// SIMATIC STEP 7 (V5.x) project Odbieranie_Kolbusy_Rob
// CPU: CPU 313C
// CPU: CPU 315-2 PN/DP
// CPU: CPU 315-2 DP
// CPU: CPU 315-2 DP
// CPU: CPU 315-2 DP
// station: Hardware
// station: Bandy
// station: P_ADR_BUS
// station: P_ADR_BUS
// station: Hardware
// station: Foliarka
// station: Hardware
// station: Odbieranie
// station: P_ADR_BUS
// station: Hardware
// station: Shuttle
// station: P_ADR_BUS
// station: P_ADR_BUS
// station: Hardware
// station: W_Help_PLC_TEST
// station: _S7H_BUSSYSTEM_CT
// station: P_ADR_BUS
// station: Configuration
// program: S7 Program
// program: S7 Program
// program: S7 Program
// program: S7 Program
// program: S7 Program(15)
// program: S7_Program_Band_Stary
// program: S7 _Bandy_1_Krew

SYMBOL_TABLE
"RUNNING_PROG"	DB 12	DB 12	// RUNNING PROGRAMME
"EDITING_PROG"	DB 13	DB 13	// EDITING PROGRAMME
"PROG_1_DATA"	DB 21	DB 21	// PROGRAMME 1
"PROG_2_DATA"	DB 22	DB 22	// PROGRAMME 2
"PROG_3_DATA"	DB 23	DB 23	// PROGRAMME 3
"PROG_4_DATA"	DB 24	DB 24	// PROGRAMME 4
"PROG_5_DATA"	DB 25	DB 25	// PROGRAMME 5
"PROG_6_DATA"	DB 26	DB 26	// PROGRAMME 6
"PROG_7_DATA"	DB 27	DB 27	// PROGRAMME 7
"PROG_8_DATA"	DB 28	DB 28	// PROGRAMME 8
"PROG_9_DATA"	DB 29	DB 29	// PROGRAMME 9
"INTERFACE_AREA"	DB 30	DB 30	// INTERFACE AREA
"MPI_GD"	DB 100	DB 100	// Blok wymiany danych po mpi
"CONTROL"	FC 1	FC 1	// CONTROL
"SAFETY_STOP"	FC 3	FC 3	// SAFETY STOP
"LAMP_TEST"	FC 4	FC 4	// LAMP TEST
"SIGNAL_OUT_CONVEYORS"	FC 5	FC 5	// EXTERNAL SIGNAL OUTPUT
"AUTOMATIC"	FC 10	FC 10	// AUTO / SEMIAUTO CHOICE
"PROGRAMME_CHOICE"	FC 11	FC 11	// START WRAPPING SEQUENCE AND PROGRAMME CHOICE
"MOTOR_TO_CLUTCH"	FC 12	FC 12	// MOTOR TO CLUTCH, SEQUENCE
"RESET_SEQ"	FC 13	FC 13	// RESET SEQUENCE
"CONVEYORING_SEQUENCE"	FC 14	FC 14	// CONVEYORING SEQUENCE
"WRAPPING_SEQUENCE"	FC 15	FC 15	// AUTOMATIC SEQUENCE
"START_AFTER_90_INFEED"	FC 16	FC 16	// START SEQ IN WRAPPING SEQ, 90 DEGREE INFEED
"90_DEGREE_INFEED"	FC 17	FC 17	// 90 DEGREE INFEED
"90_DEGREE_OUTFEED"	FC 18	FC 18	// 90 DEGREE OUTFEED
"TURN_TO/FROM_90_DEG"	FC 19	FC 19	// TURN TABLE TO/FROM 90 DEGREE
"PALLET_POS"	FC 21	FC 21	// PALLET POSITION, LENGTH MEASURE, OPTION
"TURNTABLE"	FC 22	FC 22	// TURNTABLE
"CARRIAGE"	FC 23	FC 23	// CARRIAGE
"TOPPLATE"	FC 24	FC 24	// TOPPLATE, OPTION
"FILM_FEED_SYSTEM"	FC 25	FC 25	// FILM FEED SYSTEM
"FILM_HOLDING_DEVICE"	FC 26	FC 26	// VALVES
"CUTTING_UNIT"	FC 27	FC 27	// VALVES
"HOT_AIR_WELDING"	FC 28	FC 28	// HOT AIR WELDING, OPTION
"WELDING"	FC 29	FC 29	// WELDING
"TURNTABLE_COUNTERS"	FC 32	FC 32	// TURNTABLE COUNTERS TO POSITION
"CARRIAGE_COUNTERS"	FC 33	FC 33	// CARRIAGE COUNTERS TO POSITION
"COUNTERS"	FC 34	FC 34	// COUNTERS
"CONVEYOR_1"	FC 71	FC 71	// CONVEYOR POS.1
"CONVEYOR_2"	FC 72	FC 72	// CONVEYOR AND TURN TABLE POS.2
"CONVEYOR_3"	FC 73	FC 73	// CONVEYOR POS.3
"CONVEYOR_4"	FC 74	FC 74	// CONVEYOR POS.4
"CONVEYOR_6"	FC 76	FC 76	// CONVEYOR POS.6
"CONVEYOR_7"	FC 77	FC 77	// CONVEYOR POS.7
"CONV_2"	FC 92	FC 92	// Stary przenosnik 2
"Komunikacja_GD"	FC 100	FC 100	// Komunikacja szafa foliarka
"DISPLAY_HANDLING"	FC 110	FC 110	// DISPLAY HANDLING
"MANUAL_MODE"	FC 111	FC 111	// TO RUN MACHINE IN MANUAL MODE
"ALARM"	FC 120	FC 120	// ALARM
"E 0.0"	I 0.0	BOOL	// CONTROLL VOLTAGE ON
"E 0.1"	I 0.1	BOOL	// MAIN VOLTAGE ON
"E 0.2"	I 0.2	BOOL	// TRANSDUCER TURNTABLE MOTOR FORWARD POSITION
"E 0.3"	I 0.3	BOOL	// TRANSDUCER TURNTABLE MOTOR REVERSE POSITION
"E 0.4"	I 0.4	BOOL	// TRANSDUCER TURNTABLE IN STARTPOSITION
"E 0.5"	I 0.5	BOOL	// TRANSDUCER TURNTABLE ROTATION
"E 0.6"	I 0.6	BOOL	// TRANSDUCER CARRIAGE ROTATION
"E 0.7"	I 0.7	BOOL	// TRANSDUCER TURNTABLE IN 90 DEGREE POSITION(OPTION)
"E 1.0"	I 1.0	BOOL	// TRANSDUCER PUSHER 90 DEGREE IN OUTER POSITION(OPTION)
"E 1.1"	I 1.1	BOOL	// PHOTOCELL INFEEDING START CONVEYOR
"E 1.2"	I 1.2	BOOL	// PHOTOCELL STOP INFEEDING
"E 1.3"	I 1.3	BOOL	// PHOTOCELL OUTFEEDING CONVEYOR NOT FULL(OPTION)
"E 1.5"	I 1.5	BOOL	// PHOTOCELL INDICATION PALLET 1/2 OR 1/1 SIZE OR SAFTEY
"E 1.6"	I 1.6	BOOL	// PHOTOCELL SAFETY PALLET SIZE / LENGTH MEASURE, INFEED SIDE
"E 1.7"	I 1.7	BOOL	// PHOTOCELL SAFETY PALLET SIZE / LENGTH MEASURE, OUTFEED SIDE
"E 4.0"	I 4.0	BOOL	// PB CONVEYOR 1 FORWARD(OPTION)
"E 4.1"	I 4.1	BOOL	// PB CONVEYOR 1 BACKWARD(OPTION)
"E 4.2"	I 4.2	BOOL	// PB CONVEYOR 2 FORWARD(OPTION)
"E 4.3"	I 4.3	BOOL	// PB CONVEYOR 2 BACKWARD(OPTION)
"E 4.4"	I 4.4	BOOL	// PB TURNNTABLE 2 TURN FORWARD(OPTION)
"E 4.5"	I 4.5	BOOL	// PB TURNNTABLE 2 TURN BACKWARD(OPTION)
"E 4.6"	I 4.6	BOOL	// PB CONVEYOR 3 FORWARD(OPTION)
"E 4.7"	I 4.7	BOOL	// PB CONVEYOR 3 BACKWARD(OPTION)
"E 5.0"	I 5.0	BOOL	// PB CONVEYOR 4 FORWARD
"E 5.1"	I 5.1	BOOL	// PB CONVEYOR 4 BACKWARD
"E 5.4"	I 5.4	BOOL	// PB CONVEYOR 6 FORWARD
"E 5.5"	I 5.5	BOOL	// PB CONVEYOR 6 BACKWARD
"E 5.6"	I 5.6	BOOL	// PB CONVEYOR 7 FORWARD
"E 5.7"	I 5.7	BOOL	// PB CONVEYOR 7 BACKWARD
"E 8.0"	I 8.0	BOOL	// Q PROTECTION TOP PLATE
"E 8.1"	I 8.1	BOOL	// TOPPLATE UPPER LIMIT
"E 8.2"	I 8.2	BOOL	// TOPPLATE LOWER LIMIT
"E 8.3"	I 8.3	BOOL	// TRANSDUCER TOP PLATE AGAINST GOODS
"E 8.5"	I 8.5	BOOL	// PUSH BUTTON, TOPPLATE UPWARDS
"E 8.6"	I 8.6	BOOL	// PUSH BUTTON, TOPPLATE DOWNWARDS
"E 9.0"	I 9.0	BOOL	// LS PALLET ON CONVEYOR 3(OPTION)
"E 9.1"	I 9.1	BOOL	// LS GAP MONITORING TURNTABLE CONVEYOR 3(OPTION)
"E 9.2"	I 9.2	BOOL	// LS PALLET ON CONVEYOR 1(OPTION)
"E 9.3"	I 9.3	BOOL	// LS PALLET ON CONVEYOR 2(OPTION)
"E 9.4"	I 9.4	BOOL	// AS TURN TABLE IN 0 DEGREES(OPTION)
"E 9.5"	I 9.5	BOOL	// MS SAFETY TURN TABLE IN 0 DEGREES(OPTION)
"E 9.6"	I 9.6	BOOL	// AS TURN TABLE IN 90 DEGREES(OPTION)
"E 9.7"	I 9.7	BOOL	// MS SAFETY TURN TABLE IN 90 DEGREES(OPTION)
"E 12.0"	I 12.0	BOOL	// MSI_FAULT SIGNAL
"E 12.1"	I 12.1	BOOL	// S1-S4 LIGHT  GRATING
"E 12.2"	I 12.2	BOOL	// 1.1-2.2 MSI DOORS
"E 12.3"	I 12.3	BOOL	// MSI MUTING IS ON
"E 12.4"	I 12.4	BOOL	// SIGNAL MUTING FAILURE
"E 12.5"	I 12.5	BOOL	// ALARM MUTING LAMP DEFECT
"E 12.6"	I 12.6	BOOL	// MSI RESTART BLOCKED
"E 12.7"	I 12.7	BOOL	// MSI STATE OF SAFETY OUTPUT
"E 13.0"	I 13.0	BOOL	// LS MUTING PHOTOCELL ON INFEEDING SIDE
"E 13.1"	I 13.1	BOOL	// LS MUTING PHOTOCELL ON OUTFEEDING SIDE
"E 13.2"	I 13.2	BOOL	// PB ACTIVATE SAFETY CIRCUIT
"E 13.3"	I 13.3	BOOL	// LS PALLET ON CONVEYOR 4
"E 13.4"	I 13.4	BOOL	// LS GAP MONITORING TURNTABLE CONVEYOR 6
"E 13.5"	I 13.5	BOOL	// LS PALLET ON CONVEYOR 6
"E 13.6"	I 13.6	BOOL	// LS PALLET ON CONVEYOR 7
"E 16.0"	I 16.0	BOOL	// FREQ.CONVERTER CONVEYOR 1 FAULT
"E 16.1"	I 16.1	BOOL	// FREQ.CONVERTER CONVEYOR 2 FAULT
"E 16.2"	I 16.2	BOOL	// FREQ.CONVERTER CONVEYOR 3 FAULT
"E 16.3"	I 16.3	BOOL	// FREQ.CONVERTER CONVEYOR 4 FAULT
"E 16.4"	I 16.4	BOOL	// Q MOTOR PROTECTION TURN TABLE 2 FAULT
"E 16.5"	I 16.5	BOOL	// Q MOTOR PROTECTION CONVEYOR 6 FAULT
"E 16.6"	I 16.6	BOOL	// Q MOTOR PROTECTION CONVEYOR 7 FAULT
"E 17.0"	I 17.0	BOOL	// MAIN CONTACTOR 1 ON
"E 17.1"	I 17.1	BOOL	// MAIN CONTACTOR 2 ON
"E 124.0"	I 124.0	BOOL	// PB AUTOMATIC ON
"E 124.1"	I 124.1	BOOL	// PB SEMIAUTOMATIC ON
"E 124.2"	I 124.2	BOOL	// PB STOP
"E 124.3"	I 124.3	BOOL	// PB MACHINE TO HOME POSITION / RESET
"E 124.4"	I 124.4	BOOL	// PB START SELECT WRAPPING PROGRAM
"E 124.5"	I 124.5	BOOL	// PB TURNTABLE CONVEYOR FORWARD, A
"E 124.6"	I 124.6	BOOL	// PB TURNTABLE CONVEYOR REVERSE, B
"E 124.7"	I 124.7	BOOL	// FILM CONSUMPTION (OPTION)
"E 125.0"	I 125.0	BOOL	// AS TRANSDUCER FILM END
"E 125.1"	I 125.1	BOOL	// MS CARRIAGE UPPER LIMIT
"E 125.2"	I 125.2	BOOL	// MS CARRIAGE LOWER LIMIT
"E 125.3"	I 125.3	BOOL	// AS CARRIAGE STARTPOSITION
"E 125.4"	I 125.4	BOOL	// LS PHOTOCELL PALLETHEIGHT
"E 125.5"	I 125.5	BOOL	// MS CARRIAGE CRUTSH PROTECTION
"E 125.6"	I 125.6	BOOL	// AS CUTTING DEVICE REVERSE POSITION
"E 125.7"	I 125.7	BOOL	// AS CUTTING DEVICE 1/2 - REVERSE POSITION
"E 126.0"	I 126.0	BOOL	// PROGRAMME SELECTION REMOTE COMTROLLED, BIN 1
"E 126.1"	I 126.1	BOOL	// PROGRAMME SELECTION REMOTE COMTROLLED, BIN 2
"E 126.2"	I 126.2	BOOL	// PROGRAMME SELECTION REMOTE COMTROLLED, BIN 4
"E 126.3"	I 126.3	BOOL	// FREQ.CONVERTER film motor
"E 126.4"	I 126.4	BOOL	// EXT> CONEYOR RUN IN IS RUNNING
"E 126.5"	I 126.5	BOOL	// EXT> PALLET IS READY FOR RUN IN TO CONVEYOR 1
"E 126.6"	I 126.6	BOOL	// FREQ.CONVERTER CARRIAGE FAULT
"E 126.7"	I 126.7	BOOL	// FERG.COVERTER TURN TABLE-CONVEYOR FAULT
"M 70.0"	M 70.0	BOOL	// FC71 -CONVEYOR POS.1 LOCKING
"M 70.1"	M 70.1	BOOL	// FC71 -CONVEYOR POS.1 FU FAULT
"M 70.2"	M 70.2	BOOL	// FC71 -CONVEYOR POS.1 RUN IN
"M 70.3"	M 70.3	BOOL	// FC71 -CONVEYOR POS.1 OCCUPIED
"M 70.4"	M 70.4	BOOL	// FC71 -CONVEYOR POS.1 RUN OUT
"M 70.5"	M 70.5	BOOL	// FC71 -CONVEYOR POS.1 FORWARD
"M 70.6"	M 70.6	BOOL	// FC71 -CONVEYOR POS.1 BACKWARD
"M 70.7"	M 70.7	BOOL	// FC71 -CONVEYOR POS.1 RUNTIME
"M 72.0"	M 72.0	BOOL	// FC72 -CONVEYOR POS.2 LOCKING
"M 72.1"	M 72.1	BOOL	// FC72 -CONVEYOR POS.2 FU FAULT
"M 72.2"	M 72.2	BOOL	// FC72 -CONVEYOR POS.2 RUN IN
"M 72.3"	M 72.3	BOOL	// FC72 -CONVEYOR POS.2 OCCUPIED
"M 72.4"	M 72.4	BOOL	// FC72 -CONVEYOR POS.2 RUN OUT
"M 72.5"	M 72.5	BOOL	// FC72 -CONVEYOR POS.2 FORWARD
"M 72.6"	M 72.6	BOOL	// FC72 -CONVEYOR POS.2 BACKWARD
"M 72.7"	M 72.7	BOOL	// FC72 -CONVEYOR POS.2 RUNTIME
"M 74.0"	M 74.0	BOOL	// FC72 -TURN TABLE POS.2 LOCKING
"M 74.1"	M 74.1	BOOL	// FC72 -TURN TABLE POS.2 MOTOR FAULT
"M 74.2"	M 74.2	BOOL	// FC72 -TURN TABLE POS.2 RUN TO 0DEG
"M 74.3"	M 74.3	BOOL	// FC72 -TURN TABLE POS.2 SPARE
"M 74.4"	M 74.4	BOOL	// FC72 -TURN TABLE POS.2 RUN TO 90DEG
"M 74.5"	M 74.5	BOOL	// FC72 -TURN TABLE POS.2 TURN FORWARD
"M 74.6"	M 74.6	BOOL	// FC72 -TURN TABLE POS.2 TURN BACKWARD
"M 74.7"	M 74.7	BOOL	// FC72 -TURN TABLE POS.2 RUNTIME
"M 75.0"	M 75.0	BOOL	// FC72 -TURN TABLE POS.2 GAP FAULT
"M 75.1"	M 75.1	BOOL	// FC72 -TURN TABLE POS.2 SAFETY SWITCH FAULT
"M 76.0"	M 76.0	BOOL	// FC73 -CONVEYOR POS.3 LOCKING
"M 76.1"	M 76.1	BOOL	// FC73 -CONVEYOR POS.3 FU FAULT
"M 76.2"	M 76.2	BOOL	// FC73 -CONVEYOR POS.3 RUN IN
"M 76.3"	M 76.3	BOOL	// FC73 -CONVEYOR POS.3 OCCUPIED
"M 76.4"	M 76.4	BOOL	// FC73 -CONVEYOR POS.3 RUN OUT
"M 76.5"	M 76.5	BOOL	// FC73 -CONVEYOR POS.3 FORWARD
"M 76.6"	M 76.6	BOOL	// FC73 -CONVEYOR POS.3 BACKWARD
"M 76.7"	M 76.7	BOOL	// FC73 -CONVEYOR POS.3 RUNTIME
"M 78.0"	M 78.0	BOOL	// FC74 -CONVEYOR POS.4 LOCKING
"M 78.1"	M 78.1	BOOL	// FC74 -CONVEYOR POS.4 FU FAULT
"M 78.2"	M 78.2	BOOL	// FC74 -CONVEYOR POS.4 RUN IN
"M 78.3"	M 78.3	BOOL	// FC74 -CONVEYOR POS.4 OCCUPIED
"M 78.4"	M 78.4	BOOL	// FC74 -CONVEYOR POS.4 RUN OUT
"M 78.5"	M 78.5	BOOL	// FC74 -CONVEYOR POS.4 FORWARD
"M 78.6"	M 78.6	BOOL	// FC74 -CONVEYOR POS.4 BACKWARD
"M 78.7"	M 78.7	BOOL	// FC74 -CONVEYOR POS.4 RUNTIME
"M 79.0"	M 79.0	BOOL	// FC74 -ONE SHOT RUN IN POS.4
"M 80.0"	M 80.0	BOOL	// FC76 -CONVEYOR POS.6 LOCKING
"M 80.1"	M 80.1	BOOL	// FC76 -CONVEYOR POS.6 MOTOR FAULT
"M 80.2"	M 80.2	BOOL	// FC76 -CONVEYOR POS.6 RUN IN
"M 80.3"	M 80.3	BOOL	// FC76 -CONVEYOR POS.6 OCCUPIED
"M 80.4"	M 80.4	BOOL	// FC76 -CONVEYOR POS.6 RUN OUT
"M 80.5"	M 80.5	BOOL	// FC76 -CONVEYOR POS.6 FORWARD
"M 80.6"	M 80.6	BOOL	// FC76 -CONVEYOR POS.6 BACKWARD
"M 80.7"	M 80.7	BOOL	// FC76 -CONVEYOR POS.6 RUNTIME
"M 82.0"	M 82.0	BOOL	// FC77 -CONVEYOR POS.7 LOCKING
"M 82.1"	M 82.1	BOOL	// FC77 -CONVEYOR POS.7 MOTOR FAULT
"M 82.2"	M 82.2	BOOL	// FC77 -CONVEYOR POS.7 RUN IN
"M 82.3"	M 82.3	BOOL	// FC77 -CONVEYOR POS.7 OCCUPIED
"M 82.4"	M 82.4	BOOL	// FC77 -CONVEYOR POS.7 RUN OUT
"M 82.5"	M 82.5	BOOL	// FC77 -CONVEYOR POS.7 FORWARD
"M 82.6"	M 82.6	BOOL	// FC77 -CONVEYOR POS.7 BACKWARD
"M 82.7"	M 82.7	BOOL	// FC77 -CONVEYOR POS.7 RUNTIME
"RAMP_STOP_IN_HOME_POS"	M 92.3	BOOL	// HELPMEMORY FOR RAMP DOWN BEFORE STOP IN HOME POS.
"NO_SEQ_RUNNING"	M 96.0	BOOL	// NO SEQUENCE RUNNING
"WRAPP_NOT_RUNNING"	M 96.1	BOOL	// WRAPPING PROGRAMME NOT RUNNING
"WRAPP90_NOT_RUNNING"	M 96.2	BOOL	// WRAPPING PROGRAMME FROM 90 INFEEDING NOT RUNNING
"MOTOR_TO_CLUTCH_NOT_RUN"	M 96.3	BOOL	// SEQUENCE MOTOR TO CLUTCH NOT RUNNING
"OK_FROM_TP"	M 96.5	BOOL	// TOPPLATE NOT AGAINST PALLET
"RESET_NOT_RUNNING"	M 97.2	BOOL	// RESET NOT RUNNING, MACHINE TO INITIAL POSITION
"CONVEYORING_NOT_RUNNING"	M 97.3	BOOL	// SEQUENCE CONVEYORING NOT RUNNING
"SEQ_90_INFEED_NOT_RUN"	M 97.4	BOOL	// SEQUENCE 90 DEGREE INFEEDING NOT RUNNING
"SEQ_90_OUTFEED_NOT_RUN"	M 97.5	BOOL	// SEQUENCE 90 DEGREE OUTFEEDING NOT RUNNING
"SEQ_TO/FROM_90_DEGREE"	M 97.6	BOOL	// SEQUENCE TO/FROM 90 DEGREE NOT RUNNING
"JUMP_RESET"	M 97.7	BOOL	// CONDITION TO JUMP TO RESET PROGREMME
"PULSE_PROG_REGISTER"	M 98.0	BOOL	// PULSE TO PROGRAMME REGISTER
"NO_PROG_RUNNING"	M 98.1	BOOL	// NO PROGRAMME RUNNING
"JUMP_RESET_MW"	M 98.2	BOOL	// CONDITION TO JUMP TO RESET MW, PUT ZERO TO MEM
"PULSE_RESET"	M 98.3	BOOL	// PULSE RESET
"RESET_HOLD"	M 98.4	BOOL	// PREVENT RESTART RESET SEQUENCE
"PROG_5_CHOICED"	M 98.5	BOOL	// PROGRAM 5 FILM AND OUT BACK TO STRAPPER
"PROG_4_CHOICED"	M 98.7	BOOL	// PROGRAMME 4, CONVEYORING THROUGH
"HELP_TO_M98.0"	M 99.0	BOOL	// HELP TO "PULSE_PROGRAMME REGISTER"
"HELP_TO_M98.2"	M 99.2	BOOL	// HELP TO "JUMP_RESET_MW"
"HELP_TO_M98.3"	M 99.3	BOOL	// HELP TO "PULSE_RESET"
"AUTO"	M 102.0	BOOL	// AUTOMATC MODE
"PULSE_FILMCONS"	M 103.0	BOOL	// PULSE TO COUNT UP FILM CONSUMPTION
"HELP_PULSE_FILMCONS"	M 103.1	BOOL	// HELP PULSE FILM CONSUMPTION
"COUNT_WRAP"	M 103.2	BOOL	// COUNT NUMBERS OF WRAPPING
"HELP_COUNT_WRAP"	M 103.3	BOOL	// HELP TO COUNT NUMBERS OF WRAPPING
"HELP_COUNT_FILMCON"	M 103.4	BOOL	// HELP TO COUNT FILN CONSUMPTION
"ST.MOT1"	M 118.1	BOOL	// START SEQUENCE MOTOR TO CLUTCH
"ST.MOT2"	M 118.2	BOOL	// MOTOR FORWARDS
"ST.MOT3"	M 118.3	BOOL	// MOTOR FWD SPEED 1
"ST.MOT4"	M 118.4	BOOL	// MOTOR REV SPEED 1
"ST.MOT5"	M 118.5	BOOL	// MOTOR STOP
"ST.MOT6"	M 118.6	BOOL	// TURNTABLE MOTOR IN FORWARD POSITION
"RESET_STEP1"	M 120.1	BOOL	// MOTOR BACKWARDS
"RESET_STEP2"	M 120.2	BOOL	// MOTOR SPEED 2
"RESET_STEP3"	M 120.3	BOOL	// SYNC TURNTABLE
"RESET_STEP4"	M 120.4	BOOL	// MOTOR SPEED 1
"RESET_STEP5"	M 120.5	BOOL	// MOTOR STOP, TO CLUTCH
"RESET_STEP6"	M 120.6	BOOL	// MOTOR FORWARD POSITION
"RESET_STEP7"	M 120.7	BOOL	// CARRIAGE UP
"RESET_STEP8"	M 121.0	BOOL	// CARRIAGE DOWN
"RESET_STEP9"	M 121.1	BOOL	// CARRIAGE IN POSITION
"RESET_STEP10"	M 121.2	BOOL	// RESET CYCLE FINISHED
"TPC.RES"	M 124.0	BOOL	// RESETING CONVEYOR CYCLE
"ST.TP1"	M 124.1	BOOL	// CONVEYOR INFEEDING
"ST.TP2"	M 124.2	BOOL	// OK TO START INFEEDING
"ST.TP3"	M 124.3	BOOL	// INFEEDING STOP
"ST.TP4"	M 124.4	BOOL	// OUTFEEDING REQUEST
"ST.TP5"	M 124.5	BOOL	// CONVEYOR START OUTFEEDING
"ST.TP6"	M 124.6	BOOL	// CONVEYOR OUTFEEDING
"ST.TP00"	M 124.7	BOOL	// CONVEYOR CYCLE NOT RUNNING
"FROM_LEFT"	M 126.1	BOOL	// CONVEYORING IN FROM LEFT TO RIGHT, OR FROM LEFT OUT 90
"TO_LEFT"	M 126.2	BOOL	// CONVEYORING OUT FROM RIGHT TO LEFT, OR IN 90 OUT LEFT
"FROM_RIGHT"	M 126.3	BOOL	// CONVEYORING IN FROM RIGHT TO LEFT, OR FROM RIGHT OUT 90
"TO_RIGHT"	M 126.4	BOOL	// CONVEYORING OUT FROM LEFT TO RIGHT, OR IN 90 OUT RIGHT
"FROM_90_D"	M 126.5	BOOL	// CONVEYORING IN FROM 90 DEGREE
"TO_90_D"	M 126.6	BOOL	// CONVEYORING OUT TO 90 DEGREE
"S15_SAFTY_HELP"	M 126.7	BOOL	// HELP MEM, PHOTOCELL SAFETY PALLET SIZE, TO LONG INFEEDING, 90 DEG
"PULSE_TIME_50"	M 132.0	BOOL	// BIT FOR TIME PULSE, T 50
"PALLET_INFEED"	M 132.1	BOOL	// BIT PALLET INFEEDING
"CNT_SIZE_RUN"	M 132.2	BOOL	// COUNTING SIZE IS RUNNING
"START_CNT_SIZE"	M 132.3	BOOL	// START PULSE COUNTING SIZE
"CNT_STOP_TIME"	M 132.4	BOOL	// COUNTING STOP TIME
"START_CNT_STOP_TIME"	M 132.5	BOOL	// PULSE START COUNT STOP TIME
"CNT_SIZE"	M 132.6	BOOL	// BIT FOR TIME COUNTING SIZE
"STOP_COUNTING"	M 132.7	BOOL	// BIT FOR STOP TIME COUNTING
"STOP_PALLET"	M 133.0	BOOL	// HELP BIT STOP PALLET
"STOP_SP"	M 133.6	BOOL	// STOP NEW STARTPULSE
"STOP_PST"	M 133.7	BOOL	// STOP NEW PULSE STOP TIME
"LOCK-U1"	M 134.0	BOOL	// LOCKING TURNTABLE
"TT_SPEED_LOW_FWD"	M 134.1	BOOL	// TURNTABLE SPEED LOW
"TT_SPEED_MIDDLE_FWD"	M 134.2	BOOL	// TURNTABLE SPEED MIDDLE
"TT_SPEED_HIGH"	M 134.3	BOOL	// TURNTABLE SPEED HIGH
"TT_SPEED_CONV"	M 134.4	BOOL	// CONVEYOR SPEED
"CONV_LEFT"	M 134.5	BOOL	// CONVEYOR LEFT
"CONV_RIGHT"	M 134.6	BOOL	// CONVEYOR RIGHT
"TT_FREQ_CONV_RUN"	M 134.7	BOOL
"TT_HELP_SPEED"	M 135.0	BOOL	// TURNTABLE SPEED MIDDLE OR HIGH
"TT_SPEED_LOW_REV"	M 135.1	BOOL	// TURNTABLE SPEED LOW
"TT_SPEED_MIDDLE_REV"	M 135.2	BOOL	// TURNTABLE SPEED MIDDLE
"TT_OK_TO_START"	M 135.3	BOOL	// TURNTABLE MOTOR STANDS STILL, OK TO START
"U1_INCREASE_COARSE"	M 135.4	BOOL	// TURNTABLE SPEED INCREASE COARSE
"U1_REDUSE_COARSE"	M 135.5	BOOL	// TURNTABLE SPEED REDUSE COARSE
"U1_INCREASE_FINE"	M 135.6	BOOL	// TURNTABLE SPEED INCREASE FINE
"U1_REDUSE_FINE"	M 135.7	BOOL	// TURNTABLE SPEED REDUSE FINE
"LOCK-U3"	M 136.0	BOOL	// LOCKING CARRIAGE
"CARR_SPEED_UP"	M 136.1	BOOL	// CARRIAGE SPEED UP
"CARR_SPEED_DOWN"	M 136.2	BOOL	// CARRIAGE SPEED DOWN
"CARR_HIGH_SPEED"	M 136.3	BOOL	// CARRIAGE SPEED HIGH
"CARR_RESET_SPEED"	M 136.4	BOOL	// CARRIAGE SPEED RESET
"CARR_UPWARDS"	M 136.5	BOOL	// CARRIAGE UP
"CARR_DOWNWARDS"	M 136.6	BOOL	// CARRIAGE DOWN
"CARR_FREQ_CONV_RUN"	M 136.7	BOOL
"CARR_OK_TO_START"	M 137.3	BOOL	// CARRIAGE MOTOR STANDS STILL, OK TO START
"U3_INCREASE_COARSE"	M 137.4	BOOL	// CARRIAGE SPEED INCREASE COARSE
"U3_REDUSE_COARSE"	M 137.5	BOOL	// CARRIAGE SPEED REDUSE COARSE
"U3_INCREASE_FINE"	M 137.6	BOOL	// CARRIAGE SPEED INCREASE FINE
"U3_REDUSE_FINE"	M 137.7	BOOL	// CARRIAGE SPEED REDUSE FINE
"WITH_TOPPLATE"	M 138.0	BOOL	// WRAPPING PROGRAMME WITH TOPPLATE
"TP_SAFETY_STOP_D"	M 138.1	BOOL	// TOPPLATE, SAFETY STOP DOWNWARDS
"HELP_TP_DOWNWARDS"	M 138.2	BOOL	// MEMORY TOPPLATE DOWNWARDS
"HELP_TP_UPWARDS"	M 138.3	BOOL	// MEMORY TOPPLATE UPWARDS
"LOCK-U2"	M 140.0	BOOL	// LOCKING FILM MOTOR
"FILM_FREE"	M 140.1	BOOL	// OK TO RUN FILMMOTOR
"PULSE_FFS"	M 140.2	BOOL	// PULES TO INCREASE FILMFEED VALUE
"CLUTCH_ON_CUT"	M 140.3	BOOL	// CLUTCH ON, CUTTING FILM
"ST.FF1"	M 141.1	BOOL	// INCREASE FILMFEED VALUE
"ST.FF2"	M 141.2	BOOL	// REDUCE FILMFEED VALUE
"ST.FF3"	M 141.3	BOOL	// REDUCE FILMFEED VALUE WITH FILMTENSION
"ST.FF4"	M 141.4	BOOL	// REDUCE FILMFEED AFTER CLUTCH OFF
"LOCK_VALVE"	M 142.0	BOOL	// LOCKING SOLENOIDS
"LOCK_H_A_WELD"	M 146.0	BOOL	// LOCKING HOT AIR WELDING
"HELP_TO_M146.2"	M 146.1	BOOL	// HELP TO "H A WELD START"
"H_A_WELD_START"	M 146.2	BOOL	// IMPULS HOT AIR WELDING START
"H_A_W_HEATING"	M 146.3	BOOL	// HOT AIR WELDING, HEATING
"H_A_WELD_ON"	M 146.5	BOOL	// HOT AIR WELDING ON
"H_A_WELD_FIN"	M 146.6	BOOL	// HOT AIR WELDING FINISHED
"TURNTABLE_COUNT_MEM"	M 160.0	BOOL	// COUNT UP TURNTABLE POSITION
"HELP_PF_TURNTABLE_C"	M 160.1	BOOL	// POSITIVE FLANK TURNTABLE COUNTER
"HELP_NF_TURNTABLE_C"	M 160.2	BOOL	// NEGATIVE FLANK TURNTABLE COUNTER
"OK_COMPARE"	M 160.3	BOOL
"MEM_BW"	M 160.4	BOOL	// HELP MEMORY THEN BOTTOMWRAPPING RUNNING
"MEM_TW"	M 160.5	BOOL	// HELP MEMORY THEN TOPWRAPPING RUNNING
"HELP_PF_TURNT_IN_POS"	M 160.6	BOOL	// POSITIVE FLANK TURNTABLE COUNTER
"BW_READY"	M 162.1	BOOL	// BOTTOMWRAPS READY
"TW_READY"	M 162.2	BOOL	// TOPWRAPS READY
"FILMCLAMP_OUT"	M 162.3	BOOL	// FILMCLAMP OUT TO HOME POSITION
"TT_CHANGE_TO_HIGH_SPEED"	M 162.4	BOOL	// OK TO CHANGE TURNTABLE SPEED TO HIGH
"CLUTCH_OFF"	M 162.5	BOOL	// OK TURN CLUTCH OFF
"TO_LOW_SPEED"	M 162.6	BOOL	// OK TO CHANGE TURNTABLE SPEED TO LOW
"CARR_COUNT_MEM"	M 164.0	BOOL	// COUNT UP OR DOWN CARRIAGE POSITION
"HELP_PF_CARR_C"	M 164.1	BOOL	// POSITIVE FLANK CARRIAGE COUNTER
"HELP_NF_CARR_C"	M 164.2	BOOL	// NEGATIVE FLANK CARRIAGE COUNTER
"CARR_DIRECTING"	M 164.3	BOOL	// CARRIAGE DIRECTING, 0 = DOWN, 1 = UP
"HELP_CNT_RESET_CARR"	M 164.4	BOOL
"NF_S1253"	M 164.6	BOOL	// NF "MIN POS CARR UP"
"MIN_POS_CARR_UP"	M 164.7	BOOL	// LOWERST PALLET OK TO STOP CARR, UPWARDS
"PULSE_PALLET_HIGT"	M 165.0	BOOL	// PULSE WHEN INDICATED PALLET HIGHT
"HELP_PULSE_PALLET_H"	M 165.1	BOOL	// PULSE TO READ PALLET HEIGHT
"STOP_TOP_OK"	M 165.2	BOOL	// CARRIAGE STOP AFTER PHOTOCELL
"DOWN_CUT_OK"	M 165.3	BOOL	// CARRIAGE STOP DOWNWARDS BEFORE CUTTING
"OK_TO_SYNC_TT_CONS_CARR"	M 165.4	BOOL	// OK SYNCHRONICE TURNTABLE CINSIDER CARRIAGE
"CARR_CHANGE_TO_RS"	M 165.5	BOOL	// CHANGE CARRIAGE HIGH SPEED TO RESET SPEED
"CARR_CHANGE_TO_US"	M 165.6	BOOL	// CHANGE CARRIAGE HIGH SPEED TO UP SPEED
"FRR.FC"	M 170.0	BOOL	// INTERLOCKING WRAPPING CYCLE
"ST.FC1"	M 170.1	BOOL	// START WRAPPING SEQUENCE, TOPPLATE DOWN
"ST.FC2"	M 170.2	BOOL	// MOTOR BACKWARDS, CARRIAGE DOWN
"ST.FC3"	M 170.3	BOOL	// MOTOR SPEED 2, CARRIAGE DOWN
"ST.FC4"	M 170.4	BOOL	// BOTTOMWRAPS
"ST.FC5"	M 170.5	BOOL	// CARRIAGE UP, TURNT. S.3, ARM OUT + OPEN
"ST.FC6"	M 170.6	BOOL	// CARRIAGE UP SPEED 2
"ST.FC7"	M 170.7	BOOL	// TOPPWRAPS SPEED 3
"ST.FC8"	M 171.0	BOOL	// CARRIAGE SPEED DOWNWARDS
"ST.FC9"	M 171.1	BOOL	// SYNCHRONIZE TURNTABLE
"ST.FC10"	M 171.2	BOOL	// TURNTABLE SPEED 2
"ST.FC11"	M 171.3	BOOL	// TURNTABLE SPEED 1
"ST.FC12"	M 171.4	BOOL	// TURNTABLE STOP, FILMCLAMP UP, MOTOR FORWARDS
"ST.FC13"	M 171.5	BOOL	// CUTTING DEVICE FORWARDS, CLUTCH ON
"ST.FC14"	M 171.6	BOOL	// CUTTING FILM
"ST.FC15"	M 171.7	BOOL	// CUTTING DEVICE 1/1 RETURNED
"ST.FC16"	M 172.0	BOOL	// CARRIAGE DOWN S. 3, OUTFEEDING REQUEST
"ST.FC17"	M 172.1	BOOL	// CARRIAGE DOWN RESET SPEED
"ST.FC18"	M 172.2	BOOL	// CARRIAGE STOPP
"ST.FC19"	M 172.3	BOOL	// FILMCLAMP CLOSE
"ST.FC20"	M 172.4	BOOL	// KNIFE RETURN, UPWARDS
"ST.FC21"	M 172.5	BOOL	// CUTTING DEVICE RETURN
"ST.FC22"	M 172.6	BOOL	// WRAPPING CYCLE FINISHED
"ST.90IN_1"	M 174.1	BOOL	// CUTTING DEVICE 1/2 FORWARDS
"ST.90IN_2"	M 174.2	BOOL	// KNIFE DOWNWARDS
"ST.90IN_3"	M 174.3	BOOL	// FILMCLAMP CLOSE
"ST.90IN_4"	M 174.4	BOOL	// KNIFE UPWARDS
"ST.90IN_5"	M 174.5	BOOL	// CUTTING DEVICE RETURN
"ST1_90_IN"	M 175.1	BOOL	// TURNTABLE TO 90 DEGREE
"ST2_90_IN"	M 175.2	BOOL	// INFEEDING
"ST3_90_IN"	M 175.3	BOOL	// TURNTABLE TO 0 DEGREE
"ST4_90_IN"	M 175.4	BOOL	// START WRAPPING CYCLE / P4 = SEQ FINNISHED
"ST1_90_OUT"	M 176.1	BOOL	// TURNTABLE TO 90 DEGREE, PROGRAMME 4
"ST2_90_OUT"	M 176.2	BOOL	// START OUTFEEDING 90 DEGREE
"ST3_90_OUT"	M 176.3	BOOL	// TURNTABLE TO 0 DEGREE
"ST4_90_OUT"	M 176.4	BOOL	// RESTART FILMCYCLE OR PROG 4 = SEQ FINNISHED
"ST1_TURN"	M 177.1	BOOL	// TO / FROM 0 DEGREE, MOTOR BACKWARDS
"ST2_TURN"	M 177.2	BOOL	// TO / FROM 0 DEGREE, TURNTABLE SPEED MIDDLE
"ST3_TURN"	M 177.3	BOOL	// TO / FROM 0 DEGREE, TURNTABLE SPEED LOW
"ST4_TURN"	M 177.4	BOOL	// TO / FROM 0 DEGREE, TURNTABLE STOP, MOTOR FWD
"ST5_TURN"	M 177.5	BOOL	// TO / FROM 0 DEGREE, TURNTABLE MOTOR IN POS
"TO_0_DEGREE"	M 177.6	BOOL	// HELP MEMORY TO RUN TURNTABLE TO 0 DEGREE
"TO_90_DEGREE"	M 177.7	BOOL	// HELP MEMORY TO RUN TURNTABLE TO 90 DEGREE
"Zawsze_True"	M 180.0	BOOL
"Zawsze_False"	M 180.1	BOOL
"Help_M180.2"	M 180.2	BOOL
"Help_M180.3"	M 180.3	BOOL
"Komunikacjia_OK"	M 181.0	BOOL	// Komunikacja miedzy szafa a fliarka Ok
"Help_M181.1"	M 181.1	BOOL
"Help_M182.0"	M 182.0	BOOL
"Help_M182.1"	M 182.1	BOOL
"Help_M182.2"	M 182.2	BOOL
"SUMALARM_A"	M 240.0	BOOL	// HIGHER PRIORITY
"SUMALARM_B"	M 240.1	BOOL	// LOWER PRIORITY
"MESSAGE_SHOWING"	M 240.2	BOOL	// MESSAGE SHOWING, MACHINE IN HOMEPOSITION, LAMP BLINK
"ALARM_TF"	M 240.3	BOOL	// ALARM ON TOP FILM
"SR_MEM_TO_V4_MINUS"	M 241.0	BOOL	// SR MEMORY TO Q 124.4
"HELP_TO_A23"	M 241.1	BOOL	// HELP TO ALARM A 23
"COUNT_PULSE_CHARG"	M 241.2	BOOL	// COUNT PULSE CHARGING
"HELP_COUNT_PULSE_CHARG"	M 241.3	BOOL	// HELP TO "COUNT_PULSE_CHARG"
"HELP_PF_1_HZ"	M 241.4	BOOL	// HELP TO "POSITIVE FLANK 1 HZ", M 101.5
"PF_1_HZ"	M 241.5	BOOL	// POSITIVE FLANK 1 HZ
"CONTROL_CARR_GET_STUCK"	M 241.6	BOOL	// CONTROL IF CARRIAGE HAVE BIN MOVED LAST SECOND
"CONTROL_TT_GET_STUCK"	M 241.7	BOOL	// CONTROL IF TURNTABLE HAVE BIN MOVED LAST SECOND
"A_9_GATE_OPEN"	M 242.0	BOOL	// ALARM 9, GATE OPEN
"A_10_KNIFEARM_NOT_HOME"	M 242.1	BOOL	// ALARM 10, KNIFEARM NOT IN HOME POSITION
"A_11_FILMC_TO_LONG"	M 242.2	BOOL	// ALARM 11, FILMCYCLE TIME TO LONG
"A_12_CONV_TIME_TO_LONG"	M 242.3	BOOL	// ALARM 12, CONVEYORING TIME TO LONG
"A_13_PALLET_PAUSED"	M 242.4	BOOL	// ALARM 13, PALLET PAUSED DURING INFEEDING
"A_14_LIGHT_CURTIN"	M 242.5	BOOL	// ALARM 14, SUM ALARM LIGHT CURTIN
"A_15"	M 242.6	BOOL	// ALARM 15,
"A_16"	M 242.7	BOOL	// ALARM 16,
"A_1_NOT_IN_START_POS"	M 243.0	BOOL	// ALARM 1, MACHINE NOT IN START POSITION
"A_2_FILM_END"	M 243.1	BOOL	// ALARM 2, FILM END
"A_3_OVERLOAD_CONV"	M 243.2	BOOL	// ALARM 3, OVERLOAD CONVERTER
"A_4_CARR_GET_STUCK"	M 243.3	BOOL	// ALARM 4, CARRIAGE GET STUCK
"A_5_TTABLE_GET_STUCK"	M 243.4	BOOL	// ALARM 5, TURNTABLE GET STUCK
"A_6_CLUTCH_MISSED"	M 243.5	BOOL	// ALARM 6, TURNTABLE CLUTCH MISSED
"A_7_CARR_CRUTCH_PROTECT"	M 243.6	BOOL	// ALARM 7, CARRIAGE CRUTCH PROTECTION
"A_8_MAIN_VOLTAGE_OFF"	M 243.7	BOOL	// ALARM 8, MAIN VOLTAGE OFF
"A_25_FU_CONVEYOR"	M 244.0	BOOL	// ALARM 25, FREQ.CONVERTER CONVEYOR
"A_26_MOTOR_CONVEYOR"	M 244.1	BOOL	// ALARM 26, MOTOR PROTECT.TRIPPED CONVEYOR
"A_27_GAP_TT_POS2"	M 244.2	BOOL	// ALARM 27, GAP MONITORING TT POS.2
"A_28_SAFETYSW_TT_POS2"	M 244.3	BOOL	// ALARM 28, SAFETY SWITCH TT POS.2
"A_29"	M 244.4	BOOL	// ALARM 29,
"A_30_OUTFEED_NOT_FIN"	M 244.5	BOOL	// ALARM 30, OUTFEEDING NOT FINISHED THEN INFEED STOPED
"A_31_WRONG_IN_PAR_90"	M 244.6	BOOL	// ALARM 31, WRONG IN MACHINE PARAMETERS, 2X 90 DEGREE
"A_32_WRONG_IN_PAR_PALLET"	M 244.7	BOOL	// ALARM 32, WRONG IN MACHINE PARAMETERS, 2X PALLET LENGHT
"A_17_CIRCUIT_BREAK_TRIPP"	M 245.0	BOOL	// ALARM 17, CIRCUIT BREAKER TRIPPED
"A_18_PALLET_TO_LOW"	M 245.1	BOOL	// ALARM 18, PALLET TO LOW WITH TOPPLATE
"A_19_S16_EFFECTED"	M 245.2	BOOL	// ALARM 19, S16 EFFECTED BEFORE INFEEDING
"A_20_PALLET_TO_LONG"	M 245.3	BOOL	// ALARM 20, PALLET TO LONG / WRONG POSITION
"A_21_PALLET_TO_FAR"	M 245.4	BOOL	// ALARM 21, PALLET HAS GONE TO FAR
"A_22_COUNTUR_PHOTOCELL"	M 245.5	BOOL	// ALARM 22, PALLET COUNTUR PHOTOCELL AFFECTED
"A_23"	M 245.6	BOOL	// ALARM 23
"A_24"	M 245.7	BOOL	// ALARM 24,
"M_41"	M 246.0	BOOL	// EVENT MESSAGE 41,
"M_42"	M 246.1	BOOL	// EVENT MESSAGE 42,
"M_43"	M 246.2	BOOL	// EVENT MESSAGE 43,
"M_44"	M 246.3	BOOL	// EVENT MESSAGE 44,
"M_45"	M 246.4	BOOL	// EVENT MESSAGE 45,
"M_46"	M 246.5	BOOL	// EVENT MESSAGE 46
"M_47"	M 246.6	BOOL	// EVENT MESSAGE 47,
"M_48"	M 246.7	BOOL	// EVENT MESSAGE 48,
"M_33_MACHINE_STOP"	M 247.0	BOOL	// EVENT MESSAGE 33, MACHINE STOP ACTIVATED
"M_34_CPU_BATTERY_LOW"	M 247.1	BOOL	// EVENT MESSAGE 34, CPU BATTERY LOW
"M_35"	M 247.2	BOOL	// EVENT MESSAGE 35,
"M_36"	M 247.3	BOOL	// EVENT MESSAGE 36,
"M_37"	M 247.4	BOOL	// EVENT MESSAGE 37,
"M_38"	M 247.5	BOOL	// EVENT MESSAGE 38,
"M_39"	M 247.6	BOOL	// EVENT MESSAGE 39,
"M_40"	M 247.7	BOOL	// EVENT MESSAGE 40,
"OK_RUN_BY_HAND"	M 250.0	BOOL	// OK TO RUN MACHINE BY HAND
"BY_HAND_CONV."	M 250.1	BOOL	// OK TO RUN CONVEYORING IN OR OUT BY HAND
"BY_HAND_TURNTABLE"	M 250.2	BOOL	// OK TO RUN TURNTABLE MOTOR BY HAND
"BY_HAND_CYLINDER"	M 250.3	BOOL	// OK TO RUN TT MOTOR CYLINDER BY HAND
"BY_HAND_CARRIAGE"	M 250.4	BOOL	// OK TO RUN CARRIAGE MOTOR BY HAND
"BY_HAND_TOPPLATE"	M 250.5	BOOL	// OK TO RUN TOPPLATE MOTOR BY HAND
"BY_HAND_TO/FROM_90"	M 250.6	BOOL	// OK TO RUN TURNTABLE TO / FROM 90 DEGREE
"BY_HAND_FILMMOTOR"	M 250.7	BOOL	// OK TO RUN FILMMOTOR BY HAND
"NO_RUN_BY_HAND"	M 251.0	BOOL	// NOT ABLE TO RUN BY HAND
"24V_ON"	M 252.2	BOOL	// MAIN CONTACTOR ON
"MACHINE__STOP"	M 253.0	BOOL	// MACHINE STOP, THEN OK MEM = 1
"TURNTABLE_IN_POS"	M 253.1	BOOL	// TURNTABLE IN HOMEPOSITION
"TURNTABLE_IN_90_POS"	M 253.2	BOOL	// TURNTABLE IN 90 DEGREE POSITION
"MACHINE_IN_POS"	M 253.3	BOOL	// MACHINE IN HOME POSITION A, DON´T USE
"MACHINE_IN_START_POS"	M 253.4	BOOL	// MACHINE IN HOME POSITION B, DON´T USE
"MACHINE_OK_TO_START"	M 253.5	BOOL	// MACHINE IN OK POSITION WRAPPING START
"SAFETY_OK"	M 253.7	BOOL	// SAFETY AREA OK
"M 254.0"	M 254.0	BOOL	// "0"
"10_HZ"	M 255.0	BOOL	// CLOCK PERIODS 0,1 SECONDS
"5_HZ"	M 255.1	BOOL	// CLOCK PERIODS 0,2 SECONDS
"2.5_HZ"	M 255.2	BOOL	// CLOCK PERIODS 0,4 SECONDS
"2_HZ"	M 255.3	BOOL	// CLOCK PERIODS 0,5 SECONDS
"1.25_HZ"	M 255.4	BOOL	// CLOCK PERIODS 0,8 SECONDS
"1_HZ"	M 255.5	BOOL	// CLOCK PERIODS 1,0 SECONDS
"0.625HZ"	M 255.6	BOOL	// CLOCK PERIODS 1,6 SECONDS
"0.5_HZ"	M 255.7	BOOL	// CLOCK PERIODS 2,0 SECONDS
"MD_22_RESET"	MD 22	DWORD	// RESET BITES
"MD_26_RESET"	MD 26	DWORD	// RESET BITES
"MD_30_RESET"	MD 30	DWORD	// RESET BITES
"MD_34_RESET"	MD 34	DWORD	// RESET BITES
"MD_38_RESET"	MD 38	DWORD	// RESET BITES
"MD_42_RESET"	MD 42	DWORD	// RESET BITES
"MD_46_RESET"	MD 46	DWORD	// RESET BITES
"MD_50_RESET"	MD 50	DWORD	// RESET BITES
"MD_54_RESET"	MD 54	DWORD	// RESET BITES
"MW_58_RESET"	MW 58	WORD	// RESET BITES
"MAIN_ORGANIZATION"	OB 1	OB 1	// MAIN_ORGANIZATION
"POWER_SUPPLY_FAULT"	OB 81	OB 81	// PLC BATTERY ALARM
"A 4.0"	Q 4.0	BOOL	// U2 FILMFEEDING MOTOR FORWARD
"A 4.1"	Q 4.1	BOOL	// U3 CARRIAGE MOTOR UPWARDS
"A 4.2"	Q 4.2	BOOL	// U3 CARRIAGE MOTOR DOWNWARDS
"A 4.3"	Q 4.3	BOOL	// U3 CARRIAGE MOTOR SPEED INCREASE
"A 4.4"	Q 4.4	BOOL	// U3 CARRIAGE MOTOR SPEED REDUCE
"A 4.5"	Q 4.5	BOOL	// PB AUTOMATIC
"A 4.6"	Q 4.6	BOOL	// PB SEMIAUTOMATIC
"A 4.7"	Q 4.7	BOOL	// PB MASCHINE IN START POSITION
"A 5.0"	Q 5.0	BOOL	// EXT.> / H50 REMOTE ALARMS
"A 5.1"	Q 5.1	BOOL	// EXT.> INFEEDING CONVEYOR READY FOR PALLET
"A 5.2"	Q 5.2	BOOL	// EXT.> STRETCHWRAPPER OUTFEEDING REQUEST
"A 5.3"	Q 5.3	BOOL	// EXT.> PALLET IN POSITION ON STRECHWRAPPER
"A 5.4"	Q 5.4	BOOL	// K ELECTROMAGNETIC CLUTCH
"A 5.5"	Q 5.5	BOOL	// K FILMWELDING
"A 5.6"	Q 5.6	BOOL	// K TOPPLATE UPWARDS, (OPTION)
"A 5.7"	Q 5.7	BOOL	// K TOPPLATE DOWNWARDS, (OPTION)
"A 8.0"	Q 8.0	BOOL	// K INFEEDING CONVEYOR 1 FORWARD (OPTION)
"A 8.1"	Q 8.1	BOOL	// K INFEEDING CONVEYOR 1 BACKRWARD(OPTION)
"A 8.2"	Q 8.2	BOOL	// K INFEEDING CONVEYOR 2 TURNTABLE FORWARD(OPTION)
"A 8.3"	Q 8.3	BOOL	// K INFEEDING CONVEYOR 2 TURNTABLE BACKWARD(OPTION)
"A 8.4"	Q 8.4	BOOL	// K INFEEDING CONVEYOR 3 FORWARD(OPTION)
"A 8.5"	Q 8.5	BOOL	// K INFEEDING CONVEYOR 3 BACKRWARD(OPTION)
"A 8.6"	Q 8.6	BOOL	// K INFEEDING CONVEYOR 4 FORWARD
"A 8.7"	Q 8.7	BOOL	// K INFEEDING CONVEYOR 4 BACKRWARD
"A 9.0"	Q 9.0	BOOL	// K INFEEDING CONVEYOR 1 BRAKE
"A 9.1"	Q 9.1	BOOL	// K INFEEDING CONVEYOR 2 BRAKE
"A 9.2"	Q 9.2	BOOL	// K INFEEDING CONVEYOR 3 BRAKE
"A 9.3"	Q 9.3	BOOL	// K INFEEDING CONVEYOR 4 BRAKE
"A 9.4"	Q 9.4	BOOL	// K INFEEDING TURNTABLE 2 TURN FORWARD
"A 9.5"	Q 9.5	BOOL	// K INFEEDING TURNTABLE 2 TURN BACKWARD
"A 9.7"	Q 9.7	BOOL	// LAMP SAFETY AREA OK
"A 12.0"	Q 12.0	BOOL	// K OUTFEEDING CONVEYOR 6 FORWARD
"A 12.1"	Q 12.1	BOOL	// K OUTFEEDING CONVEYOR 6 BACKRWARD
"A 12.2"	Q 12.2	BOOL	// K OUTFEEDING CONVEYOR 7 FORWARD
"A 12.3"	Q 12.3	BOOL	// K OUTFEEDING CONVEYOR 7 BACKRWARD
"A 13.0"	Q 13.0	BOOL	// ACTIVATE SAFETY AREA ( TO MSI )
"A 13.1"	Q 13.1	BOOL	// MUTING SIGNAL ON INFEEDING SIDE
"A 13.2"	Q 13.2	BOOL	// MUTING SIGNAL ON OUTFEEDING SIDE
"A 13.3"	Q 13.3	BOOL	// EXT.> CONVEYOR 4 READY FOR PALLET INFEEDING
"A 13.4"	Q 13.4	BOOL	// EXT.> PALLET IS ON CONVEYOR 4
"A 24.0"	Q 24.0	BOOL	// Y120 AIR TO HOT AIR WELDING
"A 24.1"	Q 24.1	BOOL	// K121 HEATING TO AIR WELDING
"A 124.0"	Q 124.0	BOOL	// U1 TURNTABLE MOTOR FORWARD
"A 124.1"	Q 124.1	BOOL	// U1 TURNTABLE MOTOR REVERSE
"A 124.2"	Q 124.2	BOOL	// U1 TURNTABLE MOTOR SPEED INCREASE
"A 124.3"	Q 124.3	BOOL	// U1 TURNTABLE MOTOR SPEED REDUCE
"A 124.4"	Q 124.4	BOOL	// U1 TURNTABLE ACC/DEC 2
"A 124.5"	Q 124.5	BOOL	// Y1245 TURNTABLE MOTOR BACKWARDS
"A 124.6"	Q 124.6	BOOL	// Y1246 TURNTABLE MOTOR FORWARDS
"A 124.7"	Q 124.7	BOOL	// Y1247 CUTTING DEVICE 1/2 - FORWARD
"A 125.0"	Q 125.0	BOOL	// Y1250 CUTTING DEVICE 1/1 - FORWARD
"A 125.1"	Q 125.1	BOOL	// Y1251 KNIFE
"A 125.2"	Q 125.2	BOOL	// Y1252 ARM IN
"A 125.3"	Q 125.3	BOOL	// Y1253 FILMCLAMP OPEN
"A 125.4"	Q 125.4	BOOL	// Y1254 FILMCLAMP CLOSE
"A 125.5"	Q 125.5	BOOL	// Y1255 FILMCLAMP UP
"A 125.6"	Q 125.6	BOOL	// Y1256 FILMCLAMP DOWN
"A 125.7"	Q 125.7	BOOL	// Y1257 PUSHER 90 DEGREE, OPTION
"T0_DELAY_CONV_STOP"	T 0	TIMER	// DELAY CONVEYOR STOP, PALLET IN MACHINE
"T1_OUTFEEDING_TIME"	T 1	TIMER	// PALLET OUTFEEDING TIME
"T2_DELAY_MOTOR_TO_CLUTCH"	T 2	TIMER	// DELAY START MOTOR TO CLUTCH
"T3_START_FC"	T 3	TIMER	// DELAY START FILM CYCLE
"T4_DELAY_S1254"	T 4	TIMER	// DELAY S 1254, PALLET HEIGHT
"T5_CLAMP_UP"	T 5	TIMER	// TIME BETWEEN FILMHOLDERARM MINUS AND CLAMP UP
"T6_DELAY_CUTTING"	T 6	TIMER	// TIME BETWEEN KNIFEARM PLUS AND KNIFE UP
"T7_DELAY_KNIFEARM_BACK1"	T 7	TIMER	// TIME BETWEEN KNIFE UP AND KNIFEARM MINUS TO 1/2 POS
"T8_FILMWELDING_TIME"	T 8	TIMER	// FILMWELDING TIME DURING CUTING
"T9_DELAY_CLAMP_CLOSE"	T 9	TIMER	// TIME BETWEEN KNIFE UP AND CLAMP CLOSE
"T10_DELAY_KNIFE_UP"	T 10	TIMER	// TIME BETWEEN CLAMP CLOSE AND KNIFE UP
"T11_DELAY_KNIFEARM_BACK2"	T 11	TIMER	// TIME BETWEEN KNIFE DOWN AND KNIFEARM MINUS TO HOME POS
"T12_DELAY_TT_STOP_0"	T 12	TIMER	// DELAY TIME STOP TURNTABLE IN 0 DEGREE
"T13_DELAY_TT_STOP_90"	T 13	TIMER	// DELAY TIME STOP TURNTABLE IN 90 DEGREE (FC)
"T14_DELAY_TT_S_TO_90"	T 14	TIMER	// DELAY TIME STOP TURNTABLE FROM 0 TO 90 DEGREE
"T15_DELAY_START_90"	T 15	TIMER	// DELAY TIME TO START TO/FROM 90 DEGREE
"T16_TIME_MS_90"	T 16	TIMER	// TIME TO RUN WITH MIDDLE SPEED TO/FROM 90 DEGREE
"T17_DELAT_TOPPLATE_S"	T 17	TIMER	// DELAY TOPPLATE STOP AT PALLET
"T18_FWD_TO_CLUTCH"	T 18	TIMER	// TIME MOTOR FWD TO CLUTCH
"T19_REV_TO_CLUTCH"	T 19	TIMER	// TIME MOTOR REV TO CLUTCH
"T20_RESET_=_3_SEC"	T 20	TIMER	// START RESET RING AFTER 3 SECONDS
"T21_DELAY_LAMP_TEST"	T 21	TIMER	// DELAY LAMP TEST
"T22_DELAY_LOCK_CARR"	T 22	TIMER	// DELAY LOCKING CARRIAGE
"T23_DELAY_SIGNAL_S03"	T 23	TIMER	// DELAY SIGNAL "S03 TT MOTOR REVERSE"
"T24_CARR_SPEED_ADJUST"	T 24	TIMER	// TIME TO INCREASE OR REDUCE CARRIAGE SPEED
"T25_HELP_TO_T24"	T 25	TIMER	// PAUSE TIME, HELP TO T24
"T26_TT_SPEED_ADJUST"	T 26	TIMER	// TIME TO INCREASE OR REDUCE TURNTABLE SPEED
"T27_HELP TO_T26"	T 27	TIMER	// PAUSE TIME, HELP TO T26
"T30_ONDELAY_EMERG_STOP"	T 30	TIMER	// PREVENT ALARM THEN RESET EMERGENCY_STOP
"T31_DELAY_TT_STOP_T"	T 31	TIMER	// DELAY STOP TIMER, T32, T33, T34
"T32_HAND_T12"	T 32	TIMER	// DELAY TIME STOP TURNTABLE IN 0 DEGREE
"T33_HAND_T13"	T 33	TIMER	// DELAY TIME STOP TURNTABLE IN 90 DEGREE
"T34_HAND_T14"	T 34	TIMER	// DELAY TIME STOP TURNTABLE FROM 0 TO 90 DEGREE
"T37_OPEN_DOOR"	T 37	TIMER	// TIME THEN IT´S OK TO OPEN DOOR
"T44_DELAY ALARM_22"	T 44	TIMER	// DELAY A 22: PALLET COUNTUR PHOTOCELL AFFECTED
"T50_PULSE_0.01S"	T 50	TIMER	// PULSE TIMER, 0.01 S
"T51_INFEED_L_M"	T 51	TIMER	// SAFETY TIMER FOR INFEEDING, PROTECT PULSES FROM S16
"T52_1/2_PALLET_STOP"	T 52	TIMER	// STOP TIMER CONVEYORING 1/2 PALLET
"T60_DELAY_FILMEND"	T 60	TIMER	// DELAY FILMEND ALARM (A 2)
"T61_DELAY_ALARM_10"	T 61	TIMER	// DELAY ALARM KNIFEARM NOT IN HOME POSITION
"T62_MAXTIME_FILMING"	T 62	TIMER	// MAXIMUM TIME TO RUN A SEQUENCE
"T63_MAXTIME_CONV"	T 63	TIMER	// MAXIMUM TIME CONVEYORING
"T64_DELAY_ALARM_4"	T 64	TIMER	// DELAY ALARM 4 CARRIAGE GET STUCK
"T65_DELAY_ALARM_5"	T 65	TIMER	// DELAY ALARM 5 TURNTABLE GET STUCK
"T66_MAX TIME MOTOR_CL"	T 66	TIMER	// MAX TIME MOTOR TO CLUTCH
"T67_DELAY_K2"	T 67	TIMER	// DELAY OK SIGNAL FROM K2
"T68_TT_GET_STUCK"	T 68	TIMER	// DELAY ALARM 5, TURNTABLE GET STUCK
"T69_TT_GET_STUCK"	T 69	TIMER	// DELAY ALARM 5, TURNTABLE GET STUCK
"T70_CARR_GET_STUCK"	T 70	TIMER	// DELAY ALARM 4, CARRIAGE GET STUCK
"T71_CARR_GET_STUCK"	T 71	TIMER	// DELAY ALARM 4, CARRIAGE GET STUCK
"T74_HEATING_TIME"	T 74	TIMER	// HOT AIR WELDING, HEATING TIME
"T75_WELDING_TIME"	T 75	TIMER	// HOT AIR WELDING, WELDING TIME
"T80"	T 80	TIMER	// DELAY BRIDGE UP TF
"T81"	T 81	TIMER	// DELAY START FILMFEEDING  ON PALLET
"T82"	T 82	TIMER	// DELAY STOP FILMFEEDING ON PALLET
"T83"	T 83	TIMER	// FILMLENGHT FOR FEEDING
"T84"	T 84	TIMER	// MAXIMUM  TIME FILMFEEDING
"T85"	T 85	TIMER	// DELAY STOP CONVEYOR FOR FILMCUTTING
"T86"	T 86	TIMER	// DELAY START FILMFEEDING  ON HIGH PALLET(OPTION)
"T87"	T 87	TIMER	// DELAY STOP FILMFEEDING ON HIGH PALLET(OPTION)
"T88"	T 88	TIMER	// DELAY FILM END ALARM
"T89"	T 89	TIMER	// DELAY START FILMFEEDING AFTER CUTTING
"T90"	T 90	TIMER	// DELAY SAFETY AREA OK
"T91"	T 91	TIMER	// DELAY  BRIDGE UP TF
"T92"	T 92	TIMER	// DELAY  BRAKE CONVEYOR 1
"T93"	T 93	TIMER	// DELAY  RUNTIME CONVEYOR 1
"T94"	T 94	TIMER	// DELAY  BRAKE CONVEYOR 2
"T95"	T 95	TIMER	// DELAY  RUNTIME CONVEYOR 2
"T96"	T 96	TIMER	// DELAY  RUNTIME TURN TABLE 2
"T98"	T 98	TIMER	// DELAY  BRAKE CONVEYOR 3
"T99"	T 99	TIMER	// DELAY  RUNTIME CONVEYOR 3
"T100"	T 100	TIMER	// DELAY  START PACKAGE CONVEYOR 3
"T101"	T 101	TIMER	// DELAY  BRAKE CONVEYOR 4
"T102"	T 102	TIMER	// DELAY  RUNTIME CONVEYOR 4
"T103"	T 103	TIMER	// DELAY  RUNTIME CONVEYOR 6
"T105"	T 105	TIMER	// DELAY  RUNTIME CONVEYOR 7
"T106"	T 106	TIMER	// DELAY  CONVEYOR 7 IS NOT OCCUPIED
"T 107"	T 107	TIMER	// Verzögerung Roba 7 besetzt
"T110"	T 110	TIMER	// TURNTABLE RAMP DOWN BEFORE STOP IN HOME POS.
"VAT1"	VAT 1	
"VAT2"	VAT 2	
"VAT3"	VAT 3	
"VAT4"	VAT 4	
"VAT5"	VAT 5	
"VAT6"	VAT 6	
"VAT7"	VAT 7	
"VAT8"	VAT 8	
"VAT9"	VAT 9	
"VAT10"	VAT 10	
END_SYMBOL_TABLE

FUNCTION "CONTROL" : VOID	// FC 1
TITLE = PROGRAMME SEQUENCE CONTROL
//PROJECTINFORMATION
AUTHOR : LKA
NAME : CONTROL
VERSION : 0.2
BEGIN
NETWORK
TITLE = TURNTABLE IN HOMEPOSITION
//BORD I UTGÅNGSLÄGE
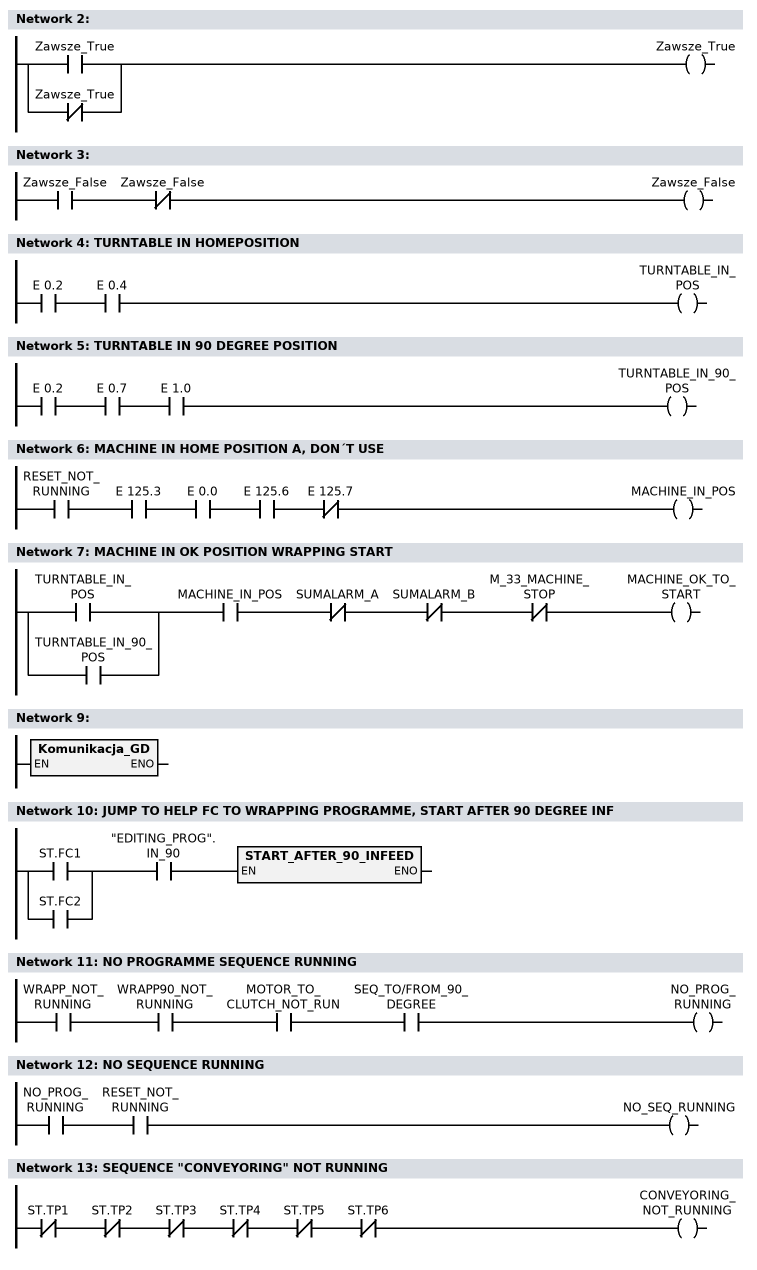
NETWORK
TITLE =
      O     "Zawsze_True";
      ON    "Zawsze_True";
      =     "Zawsze_True";
NETWORK
TITLE =
      A     "Zawsze_False";
      AN    "Zawsze_False";
      =     "Zawsze_False";
NETWORK
TITLE = TURNTABLE IN HOMEPOSITION
//BORD I UTGÅNGSLÄGE
      A     "E 0.2";
      A     "E 0.4";
      =     "TURNTABLE_IN_POS";
NETWORK
TITLE = TURNTABLE IN 90 DEGREE POSITION
//BORD I 90 GRADERS LÄGE
      A     "E 0.2";
      A     "E 0.7";
      A     "E 1.0";
      =     "TURNTABLE_IN_90_POS";
NETWORK
TITLE = MACHINE IN HOME POSITION A, DON´T USE
//MASKIN I HEMMA POS, ANVÄND EJ DENNA!!
      A     "RESET_NOT_RUNNING";
      A     "E 125.3";
      A     "E 0.0";
      A     "E 125.6";
      AN    "E 125.7";
      =     "MACHINE_IN_POS";
NETWORK
TITLE = MACHINE IN OK POSITION WRAPPING START
//MASKIN I OK POS FÖR CYKEL START
      A(;
      O     "TURNTABLE_IN_POS";
      O     "TURNTABLE_IN_90_POS";
      );
      A     "MACHINE_IN_POS";
      AN    "SUMALARM_A";
      AN    "SUMALARM_B";
      AN    "M_33_MACHINE_STOP";
      =     "MACHINE_OK_TO_START";
NETWORK
TITLE = JUMP TO WRAPPING PROGRAMME, FROM DB12.DBW8
//HOPP TILL PROGRAM ENLIGT DB12.DBW10, (PROG FUNCTION SOM SKALL KÖRAS)
      L     "RUNNING_PROG".ACTUAL_PROGRAMME;
      L     0;
      ==I;
      AN    "WRAPP90_NOT_RUNNING";
      JC    M001;
      L     "RUNNING_PROG".ACTUAL_PROGRAMME;
      L     4;
      ==I;
      JC    M001;
      CC    "WRAPPING_SEQUENCE";
M001: NOP   0;
NETWORK
TITLE =
      CALL  "Komunikacja_GD";
      NOP   0;
NETWORK
TITLE = JUMP TO HELP FC TO WRAPPING PROGRAMME, START AFTER 90 DEGREE INF
      A(;
      O     "ST.FC1";
      O     "ST.FC2";
      );
      A     "EDITING_PROG".IN_90;
      JNB   _001;
      CALL  "START_AFTER_90_INFEED";
_001: NOP   0;
NETWORK
TITLE = NO PROGRAMME SEQUENCE RUNNING
//PROGRAM SEKVENSER KÖRS EJ
      A     "WRAPP_NOT_RUNNING";
      A     "WRAPP90_NOT_RUNNING";
      A     "MOTOR_TO_CLUTCH_NOT_RUN";
      A     "SEQ_TO/FROM_90_DEGREE";
      =     "NO_PROG_RUNNING";
NETWORK
TITLE = NO SEQUENCE RUNNING
//PROGRAM ELLER RESET SEKVENSER KÖRS EJ
      A     "NO_PROG_RUNNING";
      A     "RESET_NOT_RUNNING";
      =     "NO_SEQ_RUNNING";
NETWORK
TITLE = SEQUENCE "CONVEYORING" NOT RUNNING
      AN    "ST.TP1";
      AN    "ST.TP2";
      AN    "ST.TP3";
      AN    "ST.TP4";
      AN    "ST.TP5";
      AN    "ST.TP6";
      =     "CONVEYORING_NOT_RUNNING";
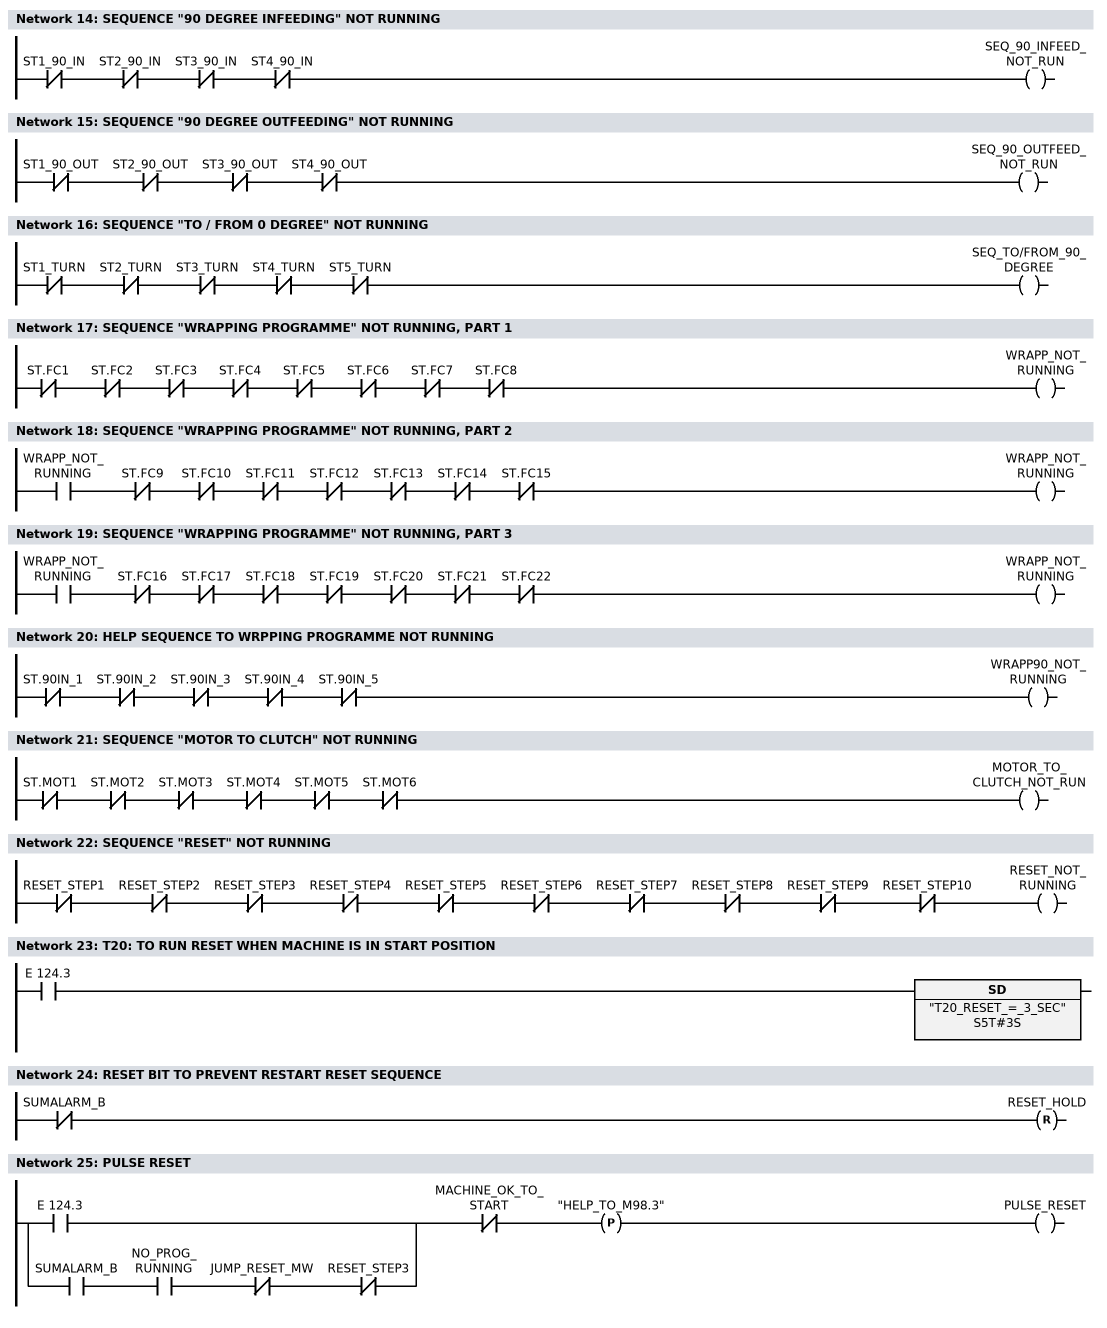
NETWORK
TITLE = SEQUENCE "90 DEGREE INFEEDING" NOT RUNNING
      AN    "ST1_90_IN";
      AN    "ST2_90_IN";
      AN    "ST3_90_IN";
      AN    "ST4_90_IN";
      =     "SEQ_90_INFEED_NOT_RUN";
NETWORK
TITLE = SEQUENCE "90 DEGREE OUTFEEDING" NOT RUNNING
      AN    "ST1_90_OUT";
      AN    "ST2_90_OUT";
      AN    "ST3_90_OUT";
      AN    "ST4_90_OUT";
      =     "SEQ_90_OUTFEED_NOT_RUN";
NETWORK
TITLE = SEQUENCE "TO / FROM 0 DEGREE" NOT RUNNING
//AVSKÄRNING PÅGÅR INTE
      AN    "ST1_TURN";
      AN    "ST2_TURN";
      AN    "ST3_TURN";
      AN    "ST4_TURN";
      AN    "ST5_TURN";
      =     "SEQ_TO/FROM_90_DEGREE";
NETWORK
TITLE = SEQUENCE "WRAPPING PROGRAMME" NOT RUNNING, PART 1
//FILM PROGRAM PÅGÅR INTE
      AN    "ST.FC1";
      AN    "ST.FC2";
      AN    "ST.FC3";
      AN    "ST.FC4";
      AN    "ST.FC5";
      AN    "ST.FC6";
      AN    "ST.FC7";
      AN    "ST.FC8";
      =     "WRAPP_NOT_RUNNING";
NETWORK
TITLE = SEQUENCE "WRAPPING PROGRAMME" NOT RUNNING, PART 2
//FILM PROGRAM PÅGÅR INTE
      A     "WRAPP_NOT_RUNNING";
      AN    "ST.FC9";
      AN    "ST.FC10";
      AN    "ST.FC11";
      AN    "ST.FC12";
      AN    "ST.FC13";
      AN    "ST.FC14";
      AN    "ST.FC15";
      =     "WRAPP_NOT_RUNNING";
NETWORK
TITLE = SEQUENCE "WRAPPING PROGRAMME" NOT RUNNING, PART 3
//FILM PROGRAM PÅGÅR INTE
      A     "WRAPP_NOT_RUNNING";
      AN    "ST.FC16";
      AN    "ST.FC17";
      AN    "ST.FC18";
      AN    "ST.FC19";
      AN    "ST.FC20";
      AN    "ST.FC21";
      AN    "ST.FC22";
      =     "WRAPP_NOT_RUNNING";
NETWORK
TITLE = HELP SEQUENCE TO WRPPING PROGRAMME NOT RUNNING
      AN    "ST.90IN_1";
      AN    "ST.90IN_2";
      AN    "ST.90IN_3";
      AN    "ST.90IN_4";
      AN    "ST.90IN_5";
      =     "WRAPP90_NOT_RUNNING";
NETWORK
TITLE = SEQUENCE "MOTOR TO CLUTCH" NOT RUNNING
      AN    "ST.MOT1";
      AN    "ST.MOT2";
      AN    "ST.MOT3";
      AN    "ST.MOT4";
      AN    "ST.MOT5";
      AN    "ST.MOT6";
      =     "MOTOR_TO_CLUTCH_NOT_RUN";
NETWORK
TITLE = SEQUENCE "RESET" NOT RUNNING
//RESET PÅGÅR INTE
      AN    "RESET_STEP1";
      AN    "RESET_STEP2";
      AN    "RESET_STEP3";
      AN    "RESET_STEP4";
      AN    "RESET_STEP5";
      AN    "RESET_STEP6";
      AN    "RESET_STEP7";
      AN    "RESET_STEP8";
      AN    "RESET_STEP9";
      AN    "RESET_STEP10";
      =     "RESET_NOT_RUNNING";
NETWORK
TITLE = T20: TO RUN RESET WHEN MACHINE IS IN START POSITION
      A     "E 124.3";
      L     S5T#3S;
      SD    "T20_RESET_=_3_SEC";
NETWORK
TITLE = RESET BIT TO PREVENT RESTART RESET SEQUENCE
      AN    "SUMALARM_B";
      R     "RESET_HOLD";
NETWORK
TITLE = PULSE RESET
      A(;
      O     "E 124.3";
      O;
      A     "SUMALARM_B";
      A     "NO_PROG_RUNNING";
      AN    "JUMP_RESET_MW";
      AN    "RESET_STEP3";
      );
      AN    "MACHINE_OK_TO_START";
      FP    "HELP_TO_M98.3";
      =     "PULSE_RESET";
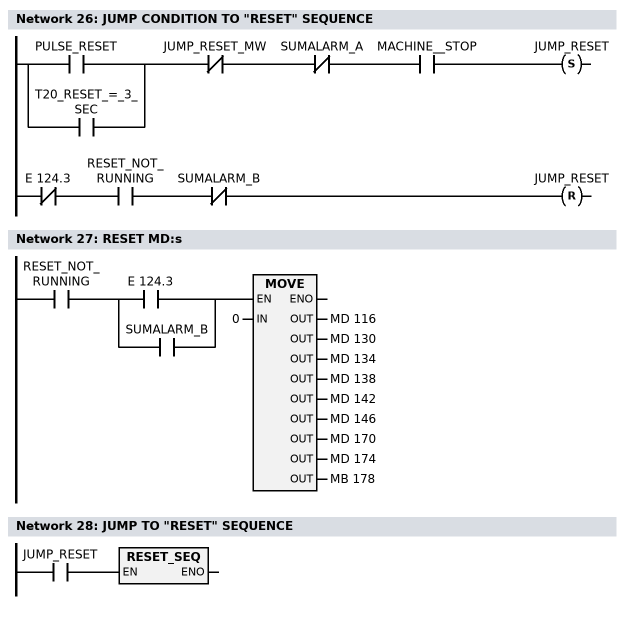
NETWORK
TITLE = JUMP CONDITION TO "RESET" SEQUENCE
      A(;
      O     "PULSE_RESET";
      O     "T20_RESET_=_3_SEC";
      );
      AN    "JUMP_RESET_MW";
      AN    "SUMALARM_A";
      A     "MACHINE__STOP";
      S     "JUMP_RESET";
      AN    "E 124.3";
      A     "RESET_NOT_RUNNING";
      AN    "SUMALARM_B";
      R     "JUMP_RESET";
      NOP   0;
NETWORK
TITLE = RESET MD:s
//första reset
      A     "RESET_NOT_RUNNING";
      A(;
      O     "E 124.3";
      O     "SUMALARM_B";
      );
      JNB   M002;
      L     0;
      T     MD 116;
      T     MD 130;
      T     MD 134;
      T     MD 138;
      T     MD 142;
      T     MD 146;
      T     MD 170;
      T     MD 174;
      T     MB 178;
M002: NOP   0;
NETWORK
TITLE = JUMP TO "RESET" SEQUENCE
//HOPP TILL RESET SEKVENS
      A     "JUMP_RESET";
      JNB   _002;
      CALL  "RESET_SEQ";
_002: NOP   0;
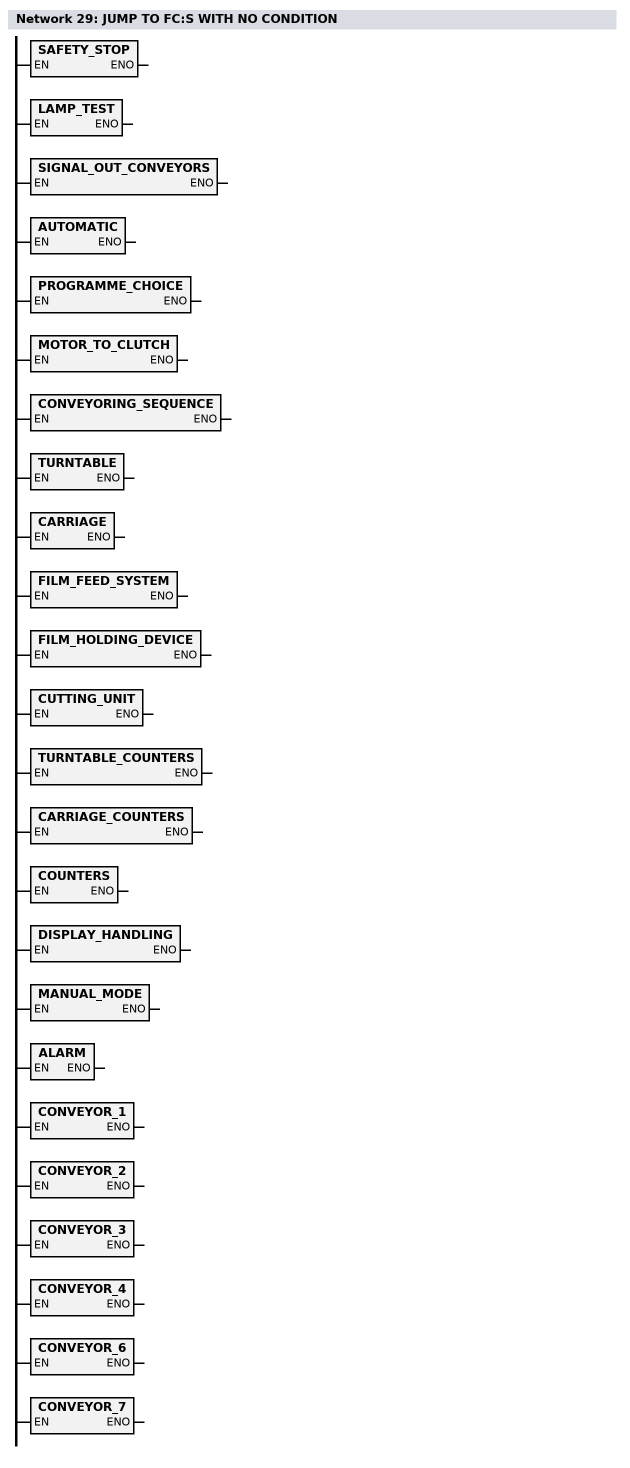
NETWORK
TITLE = JUMP TO FC:S WITH NO CONDITION
      CALL  "SAFETY_STOP";
      CALL  "LAMP_TEST";
      CALL  "SIGNAL_OUT_CONVEYORS";
      CALL  "AUTOMATIC";
      CALL  "PROGRAMME_CHOICE";
      CALL  "MOTOR_TO_CLUTCH";
      CALL  "CONVEYORING_SEQUENCE";
      CALL  "TURNTABLE";
      CALL  "CARRIAGE";
      CALL  "FILM_FEED_SYSTEM";
      CALL  "FILM_HOLDING_DEVICE";
      CALL  "CUTTING_UNIT";
      CALL  "TURNTABLE_COUNTERS";
      CALL  "CARRIAGE_COUNTERS";
      CALL  "COUNTERS";
      CALL  "DISPLAY_HANDLING";
      CALL  "MANUAL_MODE";
      CALL  "ALARM";
      CALL  "CONVEYOR_1";
      CALL  "CONVEYOR_2";
      CALL  "CONVEYOR_3";
      CALL  "CONVEYOR_4";
      CALL  "CONVEYOR_6";
      CALL  "CONVEYOR_7";
      NOP   0;
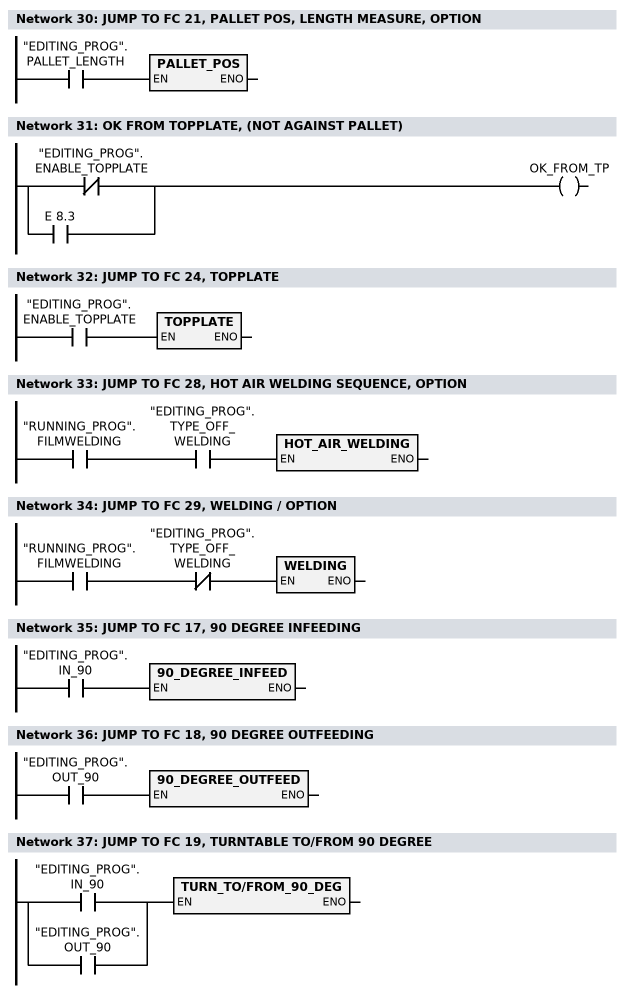
NETWORK
TITLE = JUMP TO FC 21, PALLET POS, LENGTH MEASURE, OPTION
      A     "EDITING_PROG".PALLET_LENGTH;
      JNB   _003;
      CALL  "PALLET_POS";
_003: NOP   0;
NETWORK
TITLE = OK FROM TOPPLATE, (NOT AGAINST PALLET)
      ON    "EDITING_PROG".ENABLE_TOPPLATE;
      O     "E 8.3";
      =     "OK_FROM_TP";
NETWORK
TITLE = JUMP TO FC 24, TOPPLATE
      A     "EDITING_PROG".ENABLE_TOPPLATE;
      JNB   _004;
      CALL  "TOPPLATE";
_004: NOP   0;
NETWORK
TITLE = JUMP TO FC 28, HOT AIR WELDING SEQUENCE, OPTION
      A     "RUNNING_PROG".FILMWELDING;
      A     "EDITING_PROG".TYPE_OFF_WELDING;
      JNB   _005;
      CALL  "HOT_AIR_WELDING";
_005: NOP   0;
NETWORK
TITLE = JUMP TO FC 29, WELDING / OPTION
      A     "RUNNING_PROG".FILMWELDING;
      AN    "EDITING_PROG".TYPE_OFF_WELDING;
      JNB   _006;
      CALL  "WELDING";
_006: NOP   0;
NETWORK
TITLE = JUMP TO FC 17, 90 DEGREE INFEEDING
      A     "EDITING_PROG".IN_90;
      JNB   _007;
      CALL  "90_DEGREE_INFEED";
_007: NOP   0;
NETWORK
TITLE = JUMP TO FC 18, 90 DEGREE OUTFEEDING
      A     "EDITING_PROG".OUT_90;
      JNB   _008;
      CALL  "90_DEGREE_OUTFEED";
_008: NOP   0;
NETWORK
TITLE = JUMP TO FC 19, TURNTABLE TO/FROM 90 DEGREE
      A(;
      O     "EDITING_PROG".IN_90;
      O     "EDITING_PROG".OUT_90;
      );
      JNB   _009;
      CALL  "TURN_TO/FROM_90_DEG";
_009: NOP   0;
END_FUNCTION

FUNCTION "SAFETY_STOP" : VOID	// FC 3
TITLE = SAFETY STOP
AUTHOR : LKA
NAME : SAFETY_S
VERSION : 0.1
BEGIN
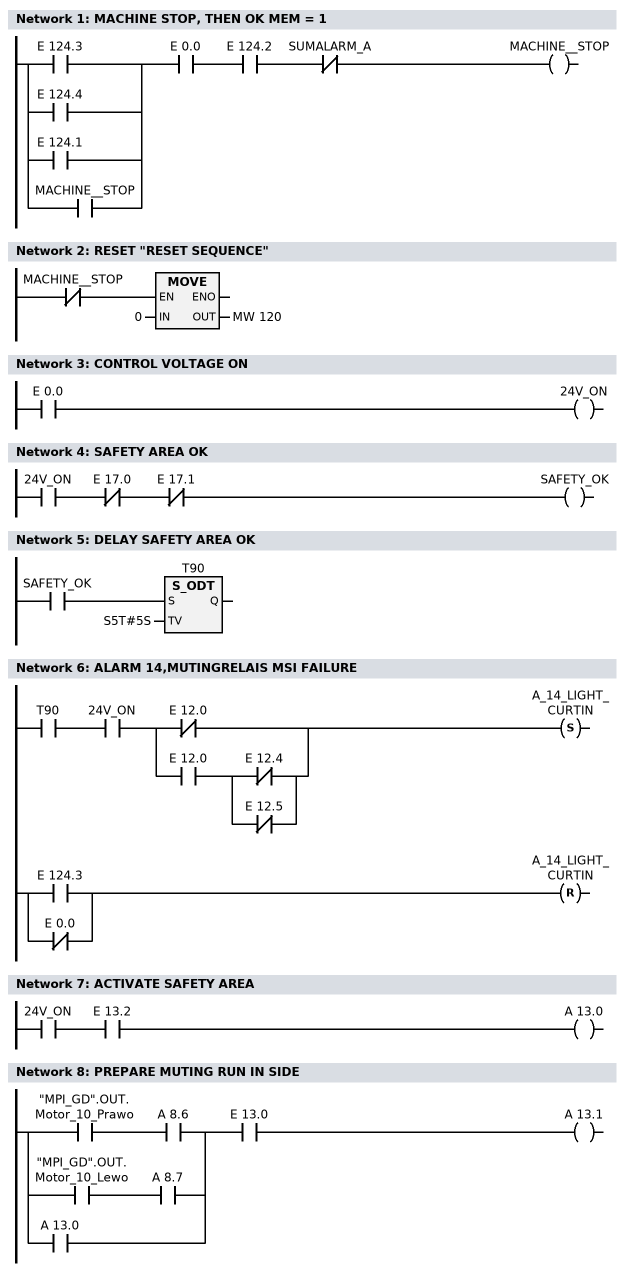
NETWORK
TITLE = MACHINE STOP, THEN OK MEM = 1
//MASKIN STOPP
      A(;
      O     "E 124.3";
      O     "E 124.4";
      O     "E 124.1";
      O     "MACHINE__STOP";
      );
      A     "E 0.0";
      A     "E 124.2";
      AN    "SUMALARM_A";
      =     "MACHINE__STOP";
NETWORK
TITLE = RESET "RESET SEQUENCE"
      AN    "MACHINE__STOP";
      JNB   _001;
      L     0;
      T     MW 120;
_001: NOP   0;
NETWORK
TITLE = CONTROL VOLTAGE ON
      A     "E 0.0";
      =     "24V_ON";
NETWORK
TITLE = SAFETY AREA OK
      A     "24V_ON";
      AN    "E 17.0";
      AN    "E 17.1";
      =     "SAFETY_OK";
NETWORK
TITLE = DELAY SAFETY AREA OK
      A     "SAFETY_OK";
      L     S5T#5S;
      SD    "T90";
      NOP   0;
      NOP   0;
      NOP   0;
      NOP   0;
NETWORK
TITLE = ALARM 14,MUTINGRELAIS MSI FAILURE
      A     "T90";
      A     "24V_ON";
      A(;
      ON    "E 12.0";
      O;
      A     "E 12.0";
      A(;
      ON    "E 12.4";
      ON    "E 12.5";
      );
      );
      S     "A_14_LIGHT_CURTIN";
      A(;
      O     "E 124.3";
      ON    "E 0.0";
      );
      R     "A_14_LIGHT_CURTIN";
      NOP   0;
NETWORK
TITLE = ACTIVATE SAFETY AREA
      A     "24V_ON";
      A     "E 13.2";
      =     "A 13.0";
NETWORK
TITLE = PREPARE MUTING RUN IN SIDE
//prawo to jest forward. Lewo to backward
      A(;
      A     "MPI_GD".OUT.Motor_10_Prawo;
      A     "A 8.6";
      O;
      A     "MPI_GD".OUT.Motor_10_Lewo;
      A     "A 8.7";
      O     "A 13.0";
      );
      A     "E 13.0";
      =     "A 13.1";
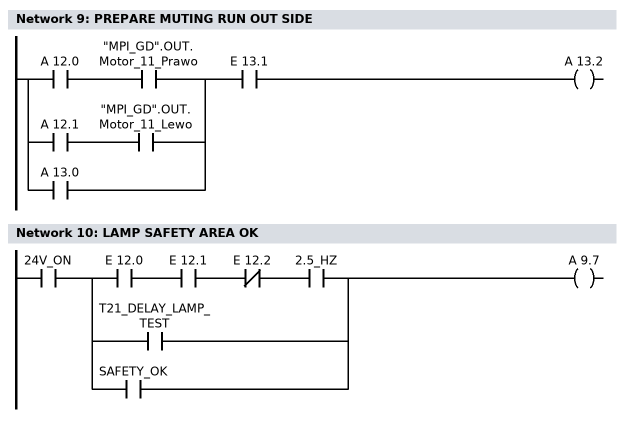
NETWORK
TITLE = PREPARE MUTING RUN OUT SIDE
      A(;
      A     "A 12.0";
      A     "MPI_GD".OUT.Motor_11_Prawo;
      O;
      A     "A 12.1";
      A     "MPI_GD".OUT.Motor_11_Lewo;
      O     "A 13.0";
      );
      A     "E 13.1";
      =     "A 13.2";
NETWORK
TITLE = LAMP SAFETY AREA OK
      A     "24V_ON";
      A(;
      A     "E 12.0";
      A     "E 12.1";
      AN    "E 12.2";
      A     "2.5_HZ";
      O     "T21_DELAY_LAMP_TEST";
      O     "SAFETY_OK";
      );
      =     "A 9.7";
END_FUNCTION

FUNCTION "LAMP_TEST" : VOID	// FC 4
TITLE = LAMP TEST
AUTHOR : LKA
NAME : LAMP_TES
VERSION : 0.1
BEGIN
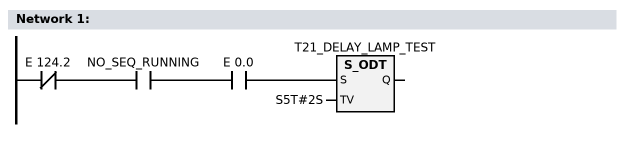
NETWORK
TITLE =
      AN    "E 124.2";
      A     "NO_SEQ_RUNNING";
      A     "E 0.0";
      L     S5T#2S;
      SD    "T21_DELAY_LAMP_TEST";
      NOP   0;
      NOP   0;
      NOP   0;
      NOP   0;
END_FUNCTION

FUNCTION "SIGNAL_OUT_CONVEYORS" : VOID	// FC 5
TITLE = SIGNAL EXCHANGES AND CONVYORS
AUTHOR : LKA
NAME : SIGNAL
VERSION : 0.1
BEGIN
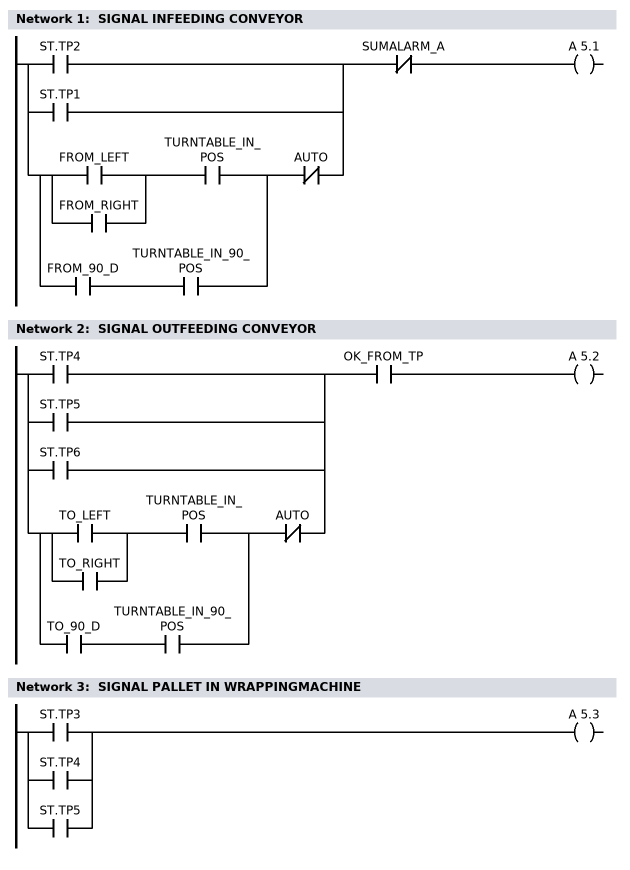
NETWORK
TITLE =  SIGNAL INFEEDING CONVEYOR
      A(;
      O     "ST.TP2";
      O     "ST.TP1";
      O;
      A(;
      A(;
      O     "FROM_LEFT";
      O     "FROM_RIGHT";
      );
      A     "TURNTABLE_IN_POS";
      O;
      A     "FROM_90_D";
      A     "TURNTABLE_IN_90_POS";
      );
      AN    "AUTO";
      );
      AN    "SUMALARM_A";
      =     "A 5.1";
NETWORK
TITLE =  SIGNAL OUTFEEDING CONVEYOR
      A(;
      O     "ST.TP4";
      O     "ST.TP5";
      O     "ST.TP6";
      O;
      A(;
      A(;
      O     "TO_LEFT";
      O     "TO_RIGHT";
      );
      A     "TURNTABLE_IN_POS";
      O;
      A     "TO_90_D";
      A     "TURNTABLE_IN_90_POS";
      );
      AN    "AUTO";
      );
      A     "OK_FROM_TP";
      =     "A 5.2";
NETWORK
TITLE =  SIGNAL PALLET IN WRAPPINGMACHINE
      O     "ST.TP3";
      O     "ST.TP4";
      O     "ST.TP5";
      =     "A 5.3";
END_FUNCTION

FUNCTION "AUTOMATIC" : VOID	// FC 10
TITLE = CONVEYORING SEQUENCE
//SEKVENS TRANSPORT, SIGNAL UTBYTE SKER HÄR
AUTHOR : LKA
NAME : AUTO
VERSION : 0.1
BEGIN
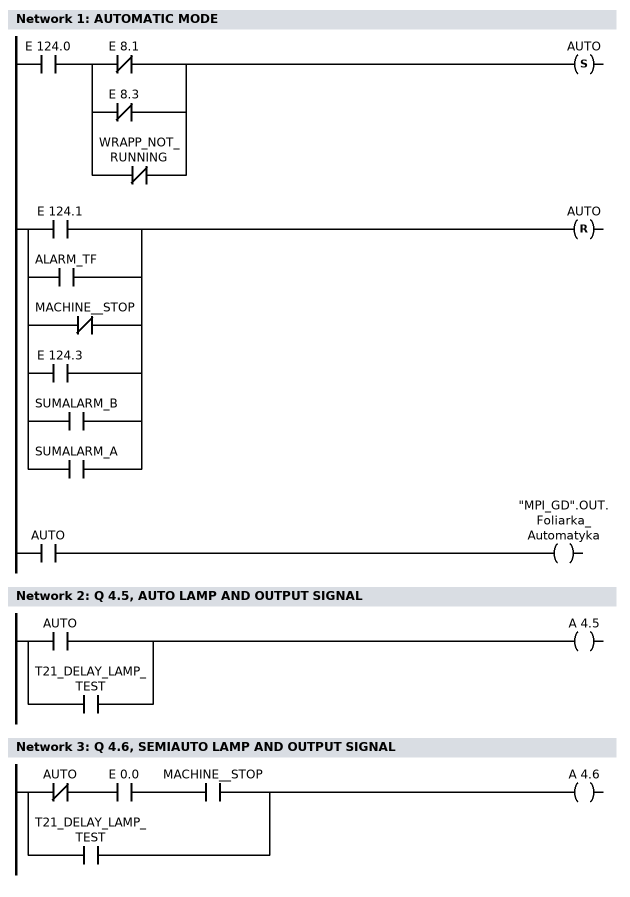
NETWORK
TITLE = AUTOMATIC MODE
      A     "E 124.0";
      A(;
      ON    "E 8.1";
      ON    "E 8.3";
      ON    "WRAPP_NOT_RUNNING";
      );
      S     "AUTO";
      A(;
      O     "E 124.1";
      O     "ALARM_TF";
      ON    "MACHINE__STOP";
      O     "E 124.3";
      O     "SUMALARM_B";
      O     "SUMALARM_A";
      );
      R     "AUTO";
      A     "AUTO";
      =     "MPI_GD".OUT.Foliarka_Automatyka;
NETWORK
TITLE = Q 4.5, AUTO LAMP AND OUTPUT SIGNAL
      O     "AUTO";
      O     "T21_DELAY_LAMP_TEST";
      =     "A 4.5";
NETWORK
TITLE = Q 4.6, SEMIAUTO LAMP AND OUTPUT SIGNAL
      AN    "AUTO";
      A     "E 0.0";
      A     "MACHINE__STOP";
      O     "T21_DELAY_LAMP_TEST";
      =     "A 4.6";
END_FUNCTION

FUNCTION "PROGRAMME_CHOICE" : VOID	// FC 11
TITLE = PROGRAMME CHOICE
AUTHOR : LKA
NAME : PROGR_C
VERSION : 0.2
BEGIN
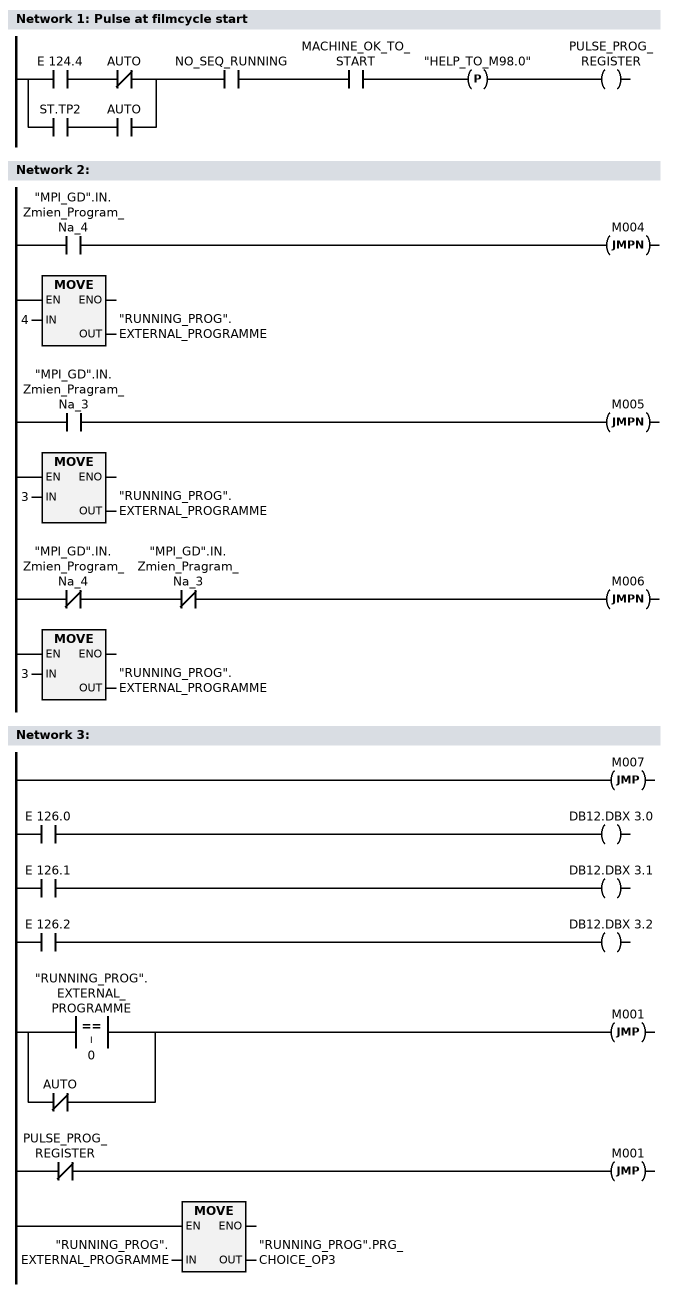
NETWORK
TITLE = Pulse at filmcycle start
//PULS VID CYKEL START
//FRÅN FC1 NW6
      A(;
      A     "E 124.4";
      AN    "AUTO";
      O;
      A     "ST.TP2";
      A     "AUTO";
      );
      A     "NO_SEQ_RUNNING";
      A     "MACHINE_OK_TO_START";
      FP    "HELP_TO_M98.0";
      =     "PULSE_PROG_REGISTER";
NETWORK
TITLE =
//|Przeslanie inforamcji o pobieraniu palety
      A     "MPI_GD".IN.Zmien_Program_Na_4;
      JCN   M004;
      L     4;
      T     "RUNNING_PROG".EXTERNAL_PROGRAMME;
M004: NOP   0;
      A     "MPI_GD".IN.Zmien_Pragram_Na_3;
      JCN   M005;
      L     3;
      T     "RUNNING_PROG".EXTERNAL_PROGRAMME;
M005: NOP   0;
      AN    "MPI_GD".IN.Zmien_Program_Na_4;
      AN    "MPI_GD".IN.Zmien_Pragram_Na_3;
      JCN   M006;
      L     3;
      T     "RUNNING_PROG".EXTERNAL_PROGRAMME;
M006: NOP   0;
NETWORK
TITLE =
//Wybor programu foliujacedgo
//zaladuj program 4
      JU    M007;
      A     "E 126.0";
      =     DB12.DBX 3.0;
      A     "E 126.1";
      =     DB12.DBX 3.1;
//zaladuj program trzeci
      A     "E 126.2";
      =     DB12.DBX 3.2;
M007: NOP   0;
      L     "RUNNING_PROG".EXTERNAL_PROGRAMME;
      L     0;
//nie laduj programow
      ==I;
      ON    "AUTO";
      JC    M001;
      AN    "PULSE_PROG_REGISTER";
      JC    M001;
      L     "RUNNING_PROG".EXTERNAL_PROGRAMME;
      T     "RUNNING_PROG".PRG_CHOICE_OP3;
M001: NOP   0;
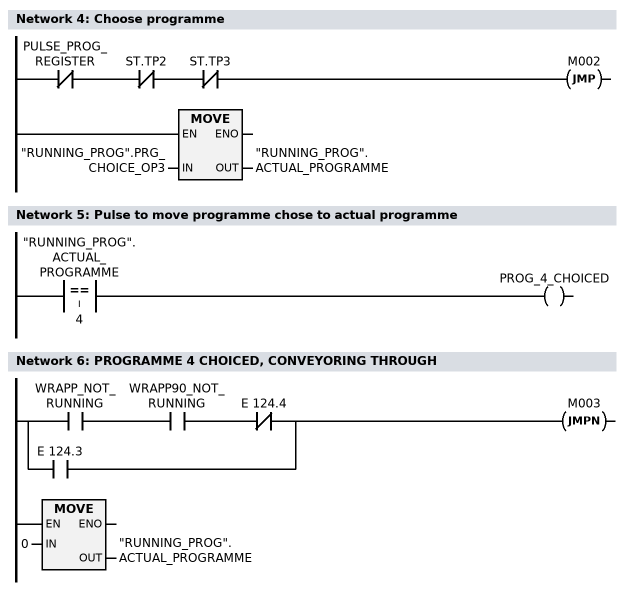
NETWORK
TITLE = Choose programme
//VÄLJ PROGRAM
//NÄR FJÄRRVAL=0 (INGA SIGNALER I8.4, I8.5, I8.6) VÄLJER MAN PROGRAM VIA OP3
//FRÅN FC110 NW 1, I HALVAUTO KAN PROGRAM VÄLJAS I OP TROTS EXTERNA PROGRAM 
//SIGNALER
      AN    "PULSE_PROG_REGISTER";
      AN    "ST.TP2";
      AN    "ST.TP3";
      JC    M002;
      L     "RUNNING_PROG".PRG_CHOICE_OP3;
      T     "RUNNING_PROG".ACTUAL_PROGRAMME;
M002: NOP   0;
NETWORK
TITLE = Pulse to move programme chose to actual programme
//PULS FLYTTA FJÄRR ELLER VALT PROGRAM TILL DB12.DBW8, (PROG SOM KÖRS)
//FRÅN FC1 NW7
//FLERA RADER RADERADE, KONTROLL OM DET FUNGERAR
      L     "RUNNING_PROG".ACTUAL_PROGRAMME;
      L     4;
      ==I;
      =     "PROG_4_CHOICED";
NETWORK
TITLE = PROGRAMME 4 CHOICED, CONVEYORING THROUGH
//FRÅN FC1 NW8
      A     "WRAPP_NOT_RUNNING";
      A     "WRAPP90_NOT_RUNNING";
      AN    "E 124.4";
      O     "E 124.3";
      JCN   M003;
      L     0;
      T     "RUNNING_PROG".ACTUAL_PROGRAMME;
M003: NOP   0;
END_FUNCTION

FUNCTION "MOTOR_TO_CLUTCH" : VOID	// FC 12
TITLE = SEQUENCE MOTOR TO CLUTCH
AUTHOR : LKA
NAME : MOTOR_TC
VERSION : 0.0
BEGIN
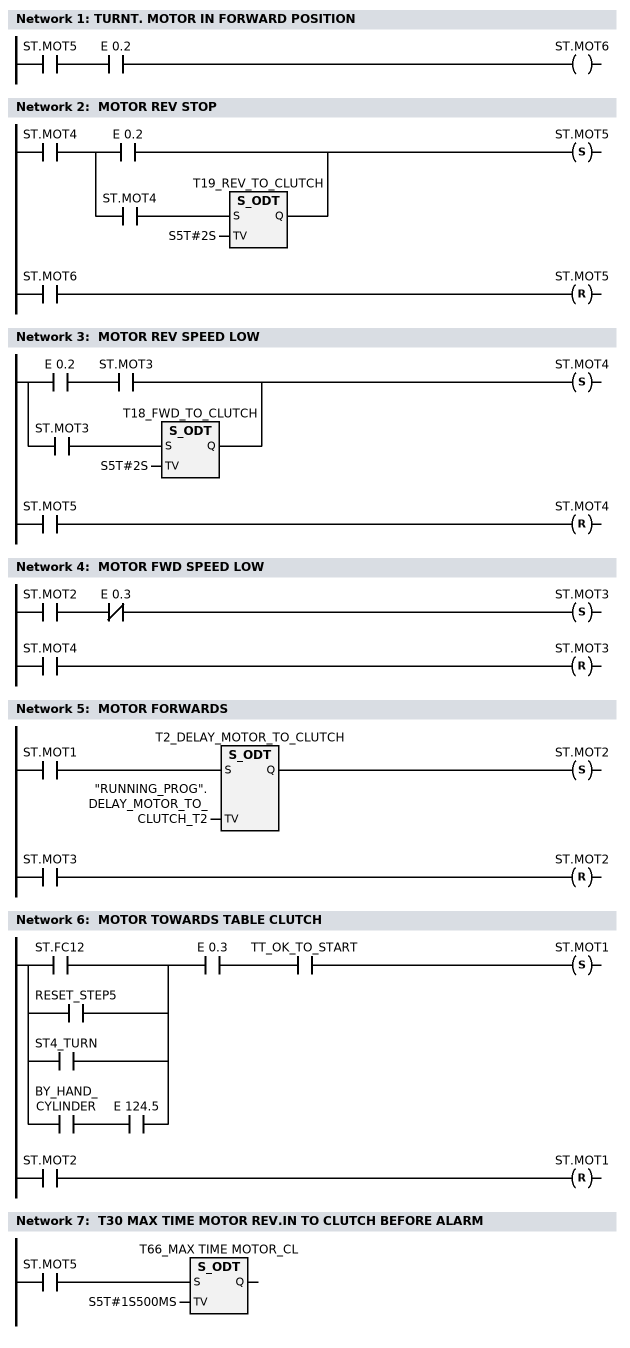
NETWORK
TITLE = TURNT. MOTOR IN FORWARD POSITION
      A     "ST.MOT5";
      A     "E 0.2";
      =     "ST.MOT6";
NETWORK
TITLE =  MOTOR REV STOP
      A     "ST.MOT4";
      A(;
      O     "E 0.2";
      O(;
      A     "ST.MOT4";
      L     S5T#2S;
      SD    "T19_REV_TO_CLUTCH";
      NOP   0;
      NOP   0;
      NOP   0;
      A     "T19_REV_TO_CLUTCH";
      );
      );
      S     "ST.MOT5";
      A     "ST.MOT6";
      R     "ST.MOT5";
      NOP   0;
NETWORK
TITLE =  MOTOR REV SPEED LOW
      A(;
      A     "E 0.2";
      A     "ST.MOT3";
      O(;
      A     "ST.MOT3";
      L     S5T#2S;
      SD    "T18_FWD_TO_CLUTCH";
      NOP   0;
      NOP   0;
      NOP   0;
      A     "T18_FWD_TO_CLUTCH";
      );
      );
      S     "ST.MOT4";
      A     "ST.MOT5";
      R     "ST.MOT4";
      NOP   0;
NETWORK
TITLE =  MOTOR FWD SPEED LOW
      A     "ST.MOT2";
      AN    "E 0.3";
      S     "ST.MOT3";
      A     "ST.MOT4";
      R     "ST.MOT3";
      NOP   0;
NETWORK
TITLE =  MOTOR FORWARDS
      A(;
      A     "ST.MOT1";
      L     "RUNNING_PROG".DELAY_MOTOR_TO_CLUTCH_T2;
      SD    "T2_DELAY_MOTOR_TO_CLUTCH";
      NOP   0;
      NOP   0;
      NOP   0;
      A     "T2_DELAY_MOTOR_TO_CLUTCH";
      );
      S     "ST.MOT2";
      A     "ST.MOT3";
      R     "ST.MOT2";
      NOP   0;
NETWORK
TITLE =  MOTOR TOWARDS TABLE CLUTCH
      A(;
      O     "ST.FC12";
      O     "RESET_STEP5";
      O     "ST4_TURN";
      O;
      A     "BY_HAND_CYLINDER";
      A     "E 124.5";
      );
      A     "E 0.3";
      A     "TT_OK_TO_START";
      S     "ST.MOT1";
      A     "ST.MOT2";
      R     "ST.MOT1";
      NOP   0;
NETWORK
TITLE =  T30 MAX TIME MOTOR REV.IN TO CLUTCH BEFORE ALARM
      A     "ST.MOT5";
      L     S5T#1S500MS;
      SD    "T66_MAX TIME MOTOR_CL";
      NOP   0;
      NOP   0;
      NOP   0;
      NOP   0;
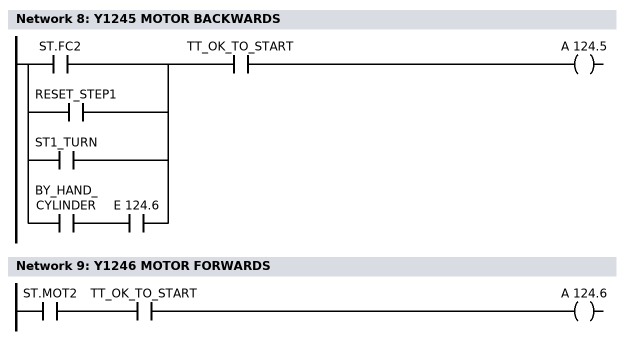
NETWORK
TITLE = Y1245 MOTOR BACKWARDS
      A(;
      O     "ST.FC2";
      O     "RESET_STEP1";
      O     "ST1_TURN";
      O;
      A     "BY_HAND_CYLINDER";
      A     "E 124.6";
      );
      A     "TT_OK_TO_START";
      =     "A 124.5";
NETWORK
TITLE = Y1246 MOTOR FORWARDS
      A     "ST.MOT2";
      A     "TT_OK_TO_START";
      =     "A 124.6";
END_FUNCTION

FUNCTION "RESET_SEQ" : VOID	// FC 13
TITLE = RESET SEKVENS
AUTHOR : LKA
NAME : RESET
VERSION : 0.2
BEGIN
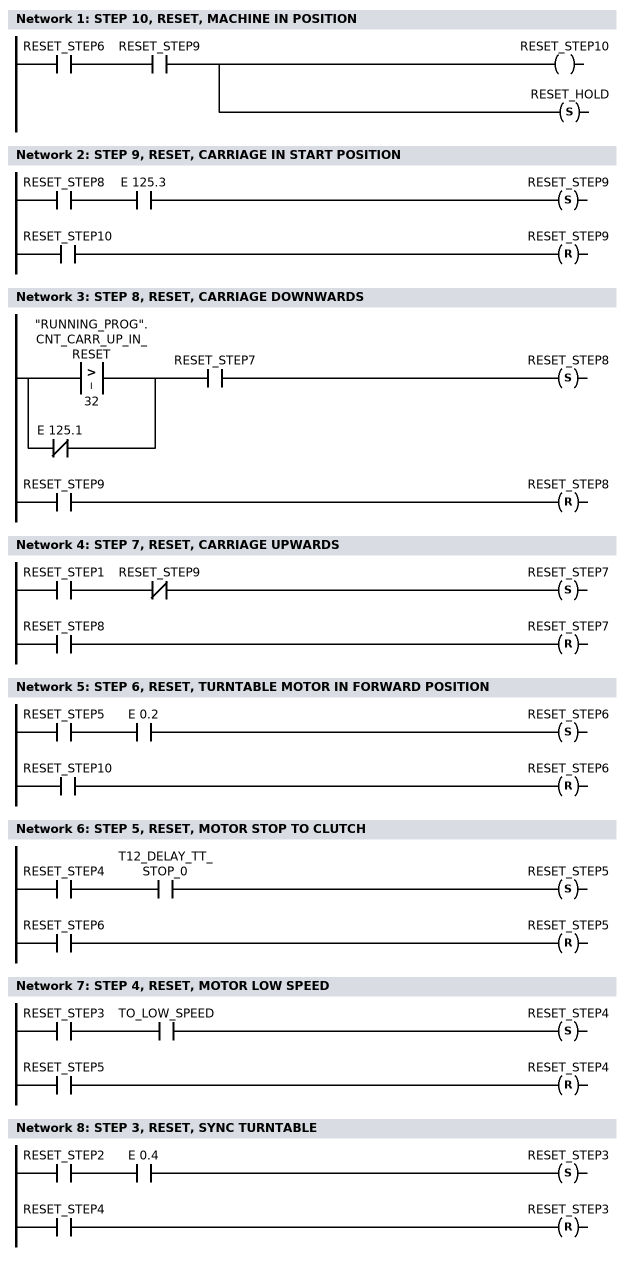
NETWORK
TITLE = STEP 10, RESET, MACHINE IN POSITION
//MASKIN I UTGÅNGSLÄGE
      A     "RESET_STEP6";
      A     "RESET_STEP9";
      =     "RESET_STEP10";
      S     "RESET_HOLD";
NETWORK
TITLE = STEP 9, RESET, CARRIAGE IN START POSITION
      A     "RESET_STEP8";
      A     "E 125.3";
      S     "RESET_STEP9";
      A     "RESET_STEP10";
      R     "RESET_STEP9";
      NOP   0;
NETWORK
TITLE = STEP 8, RESET, CARRIAGE DOWNWARDS
//HISS SKALL GÅ UPP X PULSER, RÄKNARE?????
      A(;
      O(;
      L     "RUNNING_PROG".CNT_CARR_UP_IN_RESET;
      L     32;
      >I;
      );
      ON    "E 125.1";
      );
      A     "RESET_STEP7";
      S     "RESET_STEP8";
      A     "RESET_STEP9";
      R     "RESET_STEP8";
      NOP   0;
NETWORK
TITLE = STEP 7, RESET, CARRIAGE UPWARDS
      A     "RESET_STEP1";
      AN    "RESET_STEP9";
      S     "RESET_STEP7";
      A     "RESET_STEP8";
      R     "RESET_STEP7";
      NOP   0;
NETWORK
TITLE = STEP 6, RESET, TURNTABLE MOTOR IN FORWARD POSITION
      A     "RESET_STEP5";
      A     "E 0.2";
      S     "RESET_STEP6";
      A     "RESET_STEP10";
      R     "RESET_STEP6";
      NOP   0;
NETWORK
TITLE = STEP 5, RESET, MOTOR STOP TO CLUTCH
      A     "RESET_STEP4";
      A     "T12_DELAY_TT_STOP_0";
      S     "RESET_STEP5";
      A     "RESET_STEP6";
      R     "RESET_STEP5";
      NOP   0;
NETWORK
TITLE = STEP 4, RESET, MOTOR LOW SPEED
//STEG EV BORT ????????????
      A     "RESET_STEP3";
      A     "TO_LOW_SPEED";
      S     "RESET_STEP4";
      A     "RESET_STEP5";
      R     "RESET_STEP4";
      NOP   0;
NETWORK
TITLE = STEP 3, RESET, SYNC TURNTABLE
      A     "RESET_STEP2";
      A     "E 0.4";
      S     "RESET_STEP3";
      A     "RESET_STEP4";
      R     "RESET_STEP3";
      NOP   0;
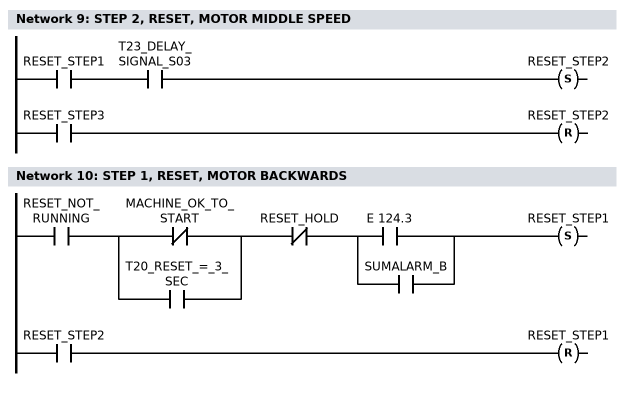
NETWORK
TITLE = STEP 2, RESET, MOTOR MIDDLE SPEED
      A     "RESET_STEP1";
      A     "T23_DELAY_SIGNAL_S03";
      S     "RESET_STEP2";
      A     "RESET_STEP3";
      R     "RESET_STEP2";
      NOP   0;
NETWORK
TITLE = STEP 1, RESET, MOTOR BACKWARDS
//OM MASKINEN EJ STÅR I UTGÅNGSLÄGE KAN SEKVENSEN STARTAS.
//KNIV NED
//FILMHÅLLARARM ÖPPNA, HEM
//AVSKÄRARENHET HEM
      A     "RESET_NOT_RUNNING";
      A(;
      ON    "MACHINE_OK_TO_START";
      O     "T20_RESET_=_3_SEC";
      );
      AN    "RESET_HOLD";
      A(;
      O     "E 124.3";
      O     "SUMALARM_B";
      );
      S     "RESET_STEP1";
      A     "RESET_STEP2";
      R     "RESET_STEP1";
      NOP   0;
END_FUNCTION

FUNCTION "CONVEYORING_SEQUENCE" : VOID	// FC 14
TITLE = CONVEYORING SEQUENCE
AUTHOR : LKA
NAME : CONVEYOR
VERSION : 0.0
BEGIN
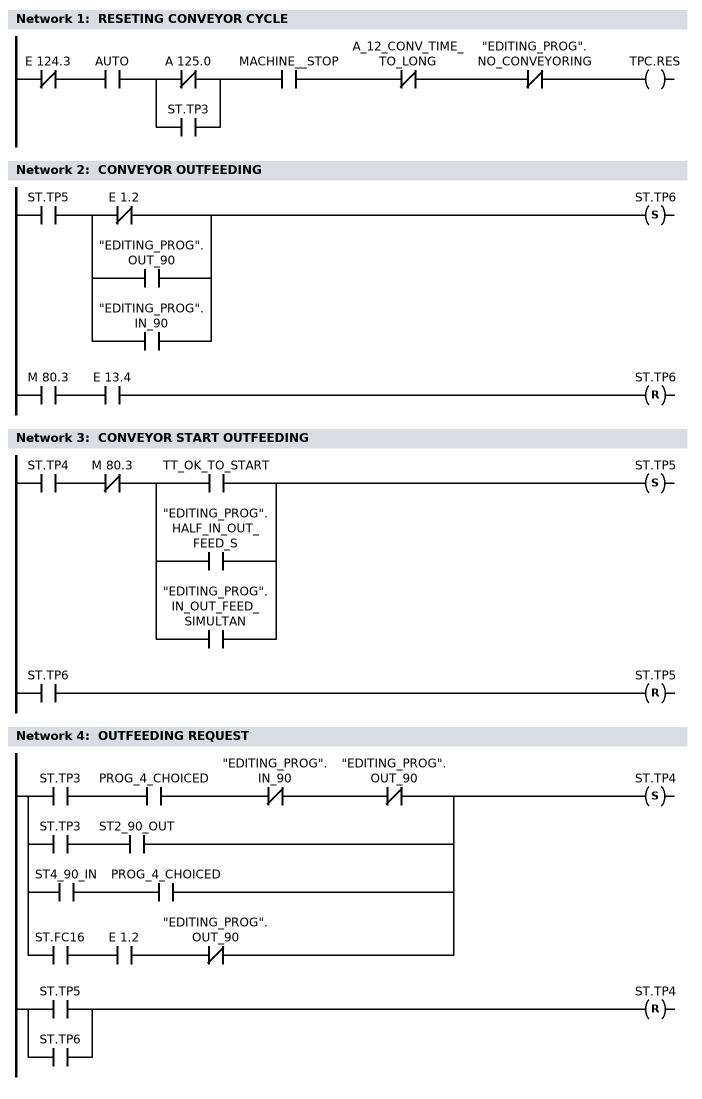
NETWORK
TITLE =  RESETING CONVEYOR CYCLE
      AN    "E 124.3";
      A     "AUTO";
      A(;
      ON    "A 125.0";
      O     "ST.TP3";
      );
      A     "MACHINE__STOP";
      AN    "A_12_CONV_TIME_TO_LONG";
      AN    "EDITING_PROG".NO_CONVEYORING;
      =     "TPC.RES";
NETWORK
TITLE =  CONVEYOR OUTFEEDING
//MER VILLKOR FÖR 90 GRADER MM.
      A     "ST.TP5";
      A(;
      ON    "E 1.2";
      O     "EDITING_PROG".OUT_90;
      O     "EDITING_PROG".IN_90;
      );
      S     "ST.TP6";
      A     "M 80.3";
      A     "E 13.4";
      R     "ST.TP6";
      NOP   0;
NETWORK
TITLE =  CONVEYOR START OUTFEEDING
      A     "ST.TP4";
      AN    "M 80.3";
      A(;
      O     "TT_OK_TO_START";
      O     "EDITING_PROG".HALF_IN_OUT_FEED_S;
      O     "EDITING_PROG".IN_OUT_FEED_SIMULTAN;
      );
      S     "ST.TP5";
      A     "ST.TP6";
      R     "ST.TP5";
      NOP   0;
NETWORK
TITLE =  OUTFEEDING REQUEST
      A(;
      A     "ST.TP3";
      A     "PROG_4_CHOICED";
      AN    "EDITING_PROG".IN_90;
      AN    "EDITING_PROG".OUT_90;
      O;
      A     "ST.TP3";
      A     "ST2_90_OUT";
      O;
      A     "ST4_90_IN";
      A     "PROG_4_CHOICED";
      O;
      A     "ST.FC16";
      A     "E 1.2";
      AN    "EDITING_PROG".OUT_90;
      );
      S     "ST.TP4";
      A(;
      O     "ST.TP5";
      O     "ST.TP6";
      );
      R     "ST.TP4";
      NOP   0;
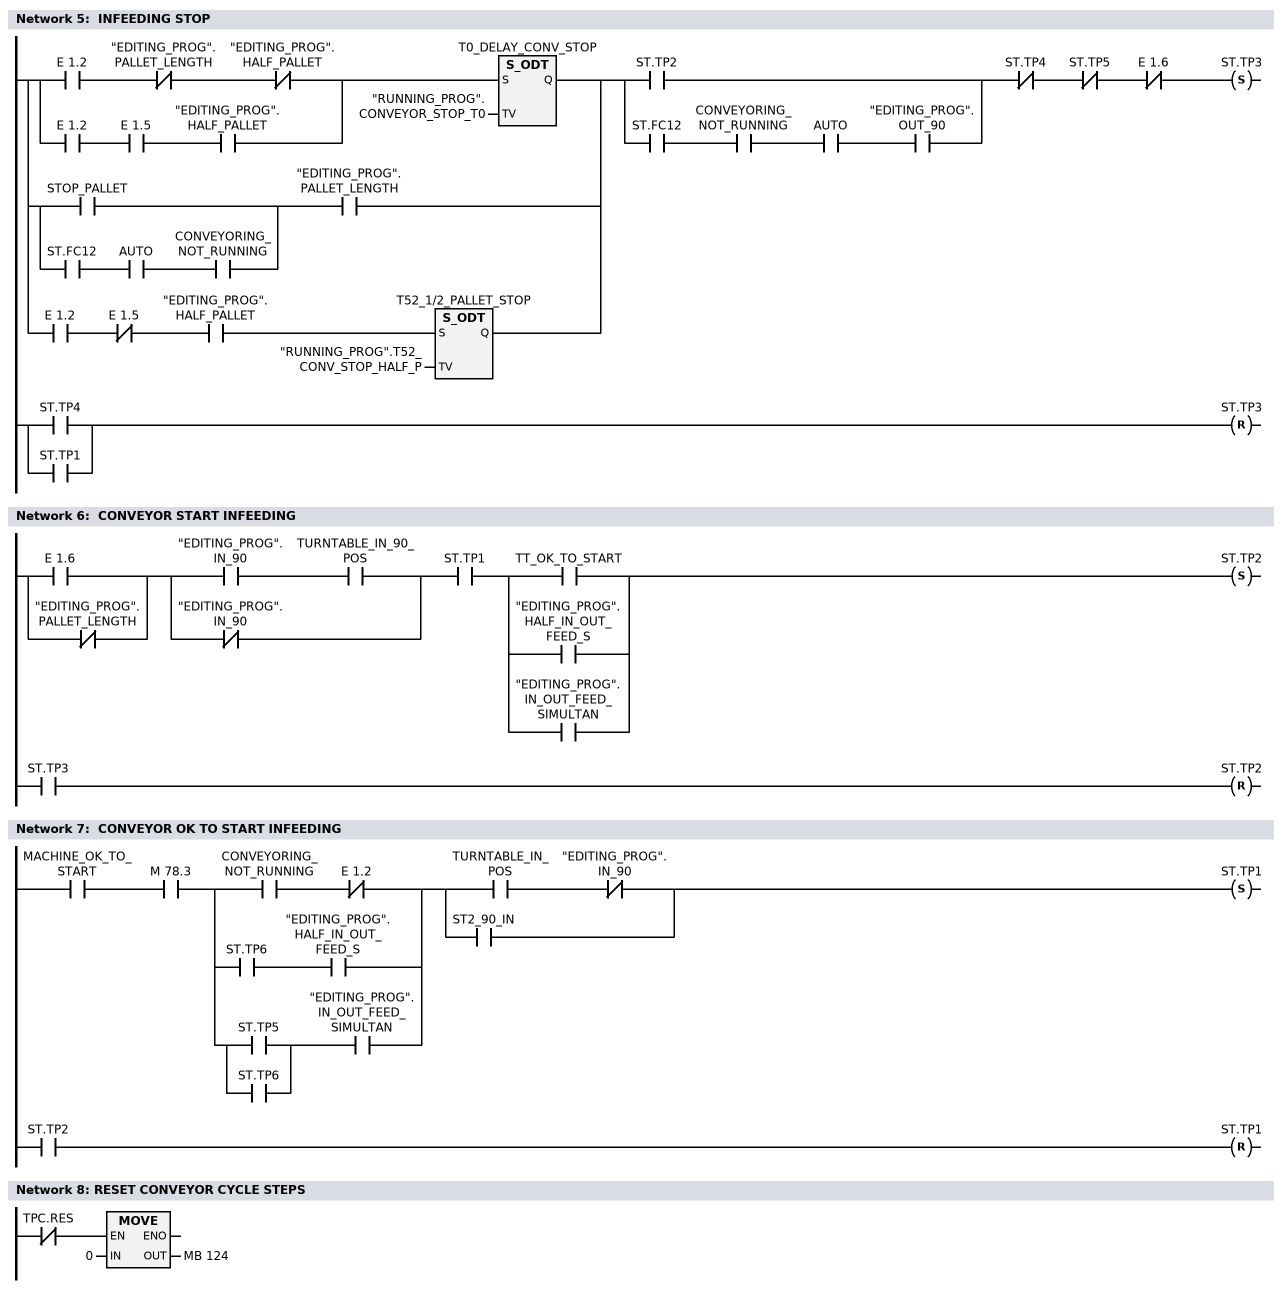
NETWORK
TITLE =  INFEEDING STOP
//bör ladda program!!!!!!
//ST-TP1 = RESET AV ST-TP3 ??????????????
      A(;
      O(;
      A(;
      A     "E 1.2";
      AN    "EDITING_PROG".PALLET_LENGTH;
      AN    "EDITING_PROG".HALF_PALLET;
      O;
      A     "E 1.2";
      A     "E 1.5";
      A     "EDITING_PROG".HALF_PALLET;
      );
      L     "RUNNING_PROG".CONVEYOR_STOP_T0;
      SD    "T0_DELAY_CONV_STOP";
      NOP   0;
      NOP   0;
      NOP   0;
      A     "T0_DELAY_CONV_STOP";
      );
      O;
      A(;
      O     "STOP_PALLET";
      O;
      A     "ST.FC12";
      A     "AUTO";
      A     "CONVEYORING_NOT_RUNNING";
      );
      A     "EDITING_PROG".PALLET_LENGTH;
      O(;
      A     "E 1.2";
      AN    "E 1.5";
      A     "EDITING_PROG".HALF_PALLET;
      L     "RUNNING_PROG".T52_CONV_STOP_HALF_P;
      SD    "T52_1/2_PALLET_STOP";
      NOP   0;
      NOP   0;
      NOP   0;
      A     "T52_1/2_PALLET_STOP";
      );
      );
      A(;
      O     "ST.TP2";
      O;
      A     "ST.FC12";
      A     "CONVEYORING_NOT_RUNNING";
      A     "AUTO";
      A     "EDITING_PROG".OUT_90;
      );
      AN    "ST.TP4";
      AN    "ST.TP5";
      AN    "E 1.6";
      S     "ST.TP3";
      A(;
      O     "ST.TP4";
      O     "ST.TP1";
      );
      R     "ST.TP3";
      NOP   0;
NETWORK
TITLE =  CONVEYOR START INFEEDING
      A(;
      O     "E 1.6";
      ON    "EDITING_PROG".PALLET_LENGTH;
      );
      A(;
      A     "EDITING_PROG".IN_90;
      A     "TURNTABLE_IN_90_POS";
      ON    "EDITING_PROG".IN_90;
      );
      A     "ST.TP1";
      A(;
      O     "TT_OK_TO_START";
      O     "EDITING_PROG".HALF_IN_OUT_FEED_S;
      O     "EDITING_PROG".IN_OUT_FEED_SIMULTAN;
      );
      S     "ST.TP2";
      A     "ST.TP3";
      R     "ST.TP2";
      NOP   0;
NETWORK
TITLE =  CONVEYOR OK TO START INFEEDING
      A     "MACHINE_OK_TO_START";
      A     "M 78.3";
      A(;
      A     "CONVEYORING_NOT_RUNNING";
      AN    "E 1.2";
      O;
      A     "ST.TP6";
      A     "EDITING_PROG".HALF_IN_OUT_FEED_S;
      O;
      A(;
      O     "ST.TP5";
      O     "ST.TP6";
      );
      A     "EDITING_PROG".IN_OUT_FEED_SIMULTAN;
      );
      A(;
      A     "TURNTABLE_IN_POS";
      AN    "EDITING_PROG".IN_90;
      O     "ST2_90_IN";
      );
      S     "ST.TP1";
      A     "ST.TP2";
      R     "ST.TP1";
      NOP   0;
NETWORK
TITLE = RESET CONVEYOR CYCLE STEPS
      AN    "TPC.RES";
      JNB   _001;
      L     0;
      T     MB 124;
_001: NOP   0;
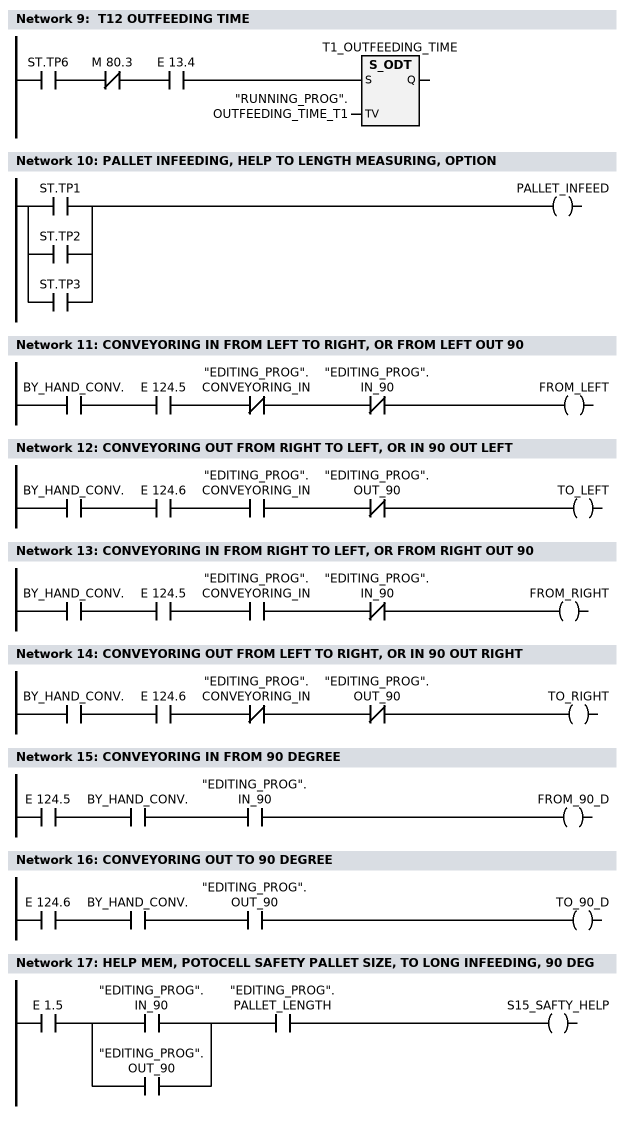
NETWORK
TITLE =  T12 OUTFEEDING TIME
//S14 BYGLAS NÄR BARA TVÅ SIGNALER IN FINNS!
      A     "ST.TP6";
      AN    "M 80.3";
      A     "E 13.4";
      L     "RUNNING_PROG".OUTFEEDING_TIME_T1;
      SD    "T1_OUTFEEDING_TIME";
      NOP   0;
      NOP   0;
      NOP   0;
      NOP   0;
NETWORK
TITLE = PALLET INFEEDING, HELP TO LENGTH MEASURING, OPTION
      O     "ST.TP1";
      O     "ST.TP2";
      O     "ST.TP3";
      =     "PALLET_INFEED";
NETWORK
TITLE = CONVEYORING IN FROM LEFT TO RIGHT, OR FROM LEFT OUT 90
      A     "BY_HAND_CONV.";
      A     "E 124.5";
      AN    "EDITING_PROG".CONVEYORING_IN;
      AN    "EDITING_PROG".IN_90;
      =     "FROM_LEFT";
NETWORK
TITLE = CONVEYORING OUT FROM RIGHT TO LEFT, OR IN 90 OUT LEFT
      A     "BY_HAND_CONV.";
      A     "E 124.6";
      A     "EDITING_PROG".CONVEYORING_IN;
      AN    "EDITING_PROG".OUT_90;
      =     "TO_LEFT";
NETWORK
TITLE = CONVEYORING IN FROM RIGHT TO LEFT, OR FROM RIGHT OUT 90
      A     "BY_HAND_CONV.";
      A     "E 124.5";
      A     "EDITING_PROG".CONVEYORING_IN;
      AN    "EDITING_PROG".IN_90;
      =     "FROM_RIGHT";
NETWORK
TITLE = CONVEYORING OUT FROM LEFT TO RIGHT, OR IN 90 OUT RIGHT
      A     "BY_HAND_CONV.";
      A     "E 124.6";
      AN    "EDITING_PROG".CONVEYORING_IN;
      AN    "EDITING_PROG".OUT_90;
      =     "TO_RIGHT";
NETWORK
TITLE = CONVEYORING IN FROM 90 DEGREE
      A     "E 124.5";
      A     "BY_HAND_CONV.";
      A     "EDITING_PROG".IN_90;
      =     "FROM_90_D";
NETWORK
TITLE = CONVEYORING OUT TO 90 DEGREE
      A     "E 124.6";
      A     "BY_HAND_CONV.";
      A     "EDITING_PROG".OUT_90;
      =     "TO_90_D";
NETWORK
TITLE = HELP MEM, POTOCELL SAFETY PALLET SIZE, TO LONG INFEEDING, 90 DEG
      A     "E 1.5";
      A(;
      O     "EDITING_PROG".IN_90;
      O     "EDITING_PROG".OUT_90;
      );
      A     "EDITING_PROG".PALLET_LENGTH;
      =     "S15_SAFTY_HELP";
END_FUNCTION

FUNCTION "WRAPPING_SEQUENCE" : VOID	// FC 15
TITLE = WRAPPING SEQUENCE, (FILM CYCLE)
AUTHOR : LKA
NAME : WRAPSEQ
VERSION : 0.0
BEGIN
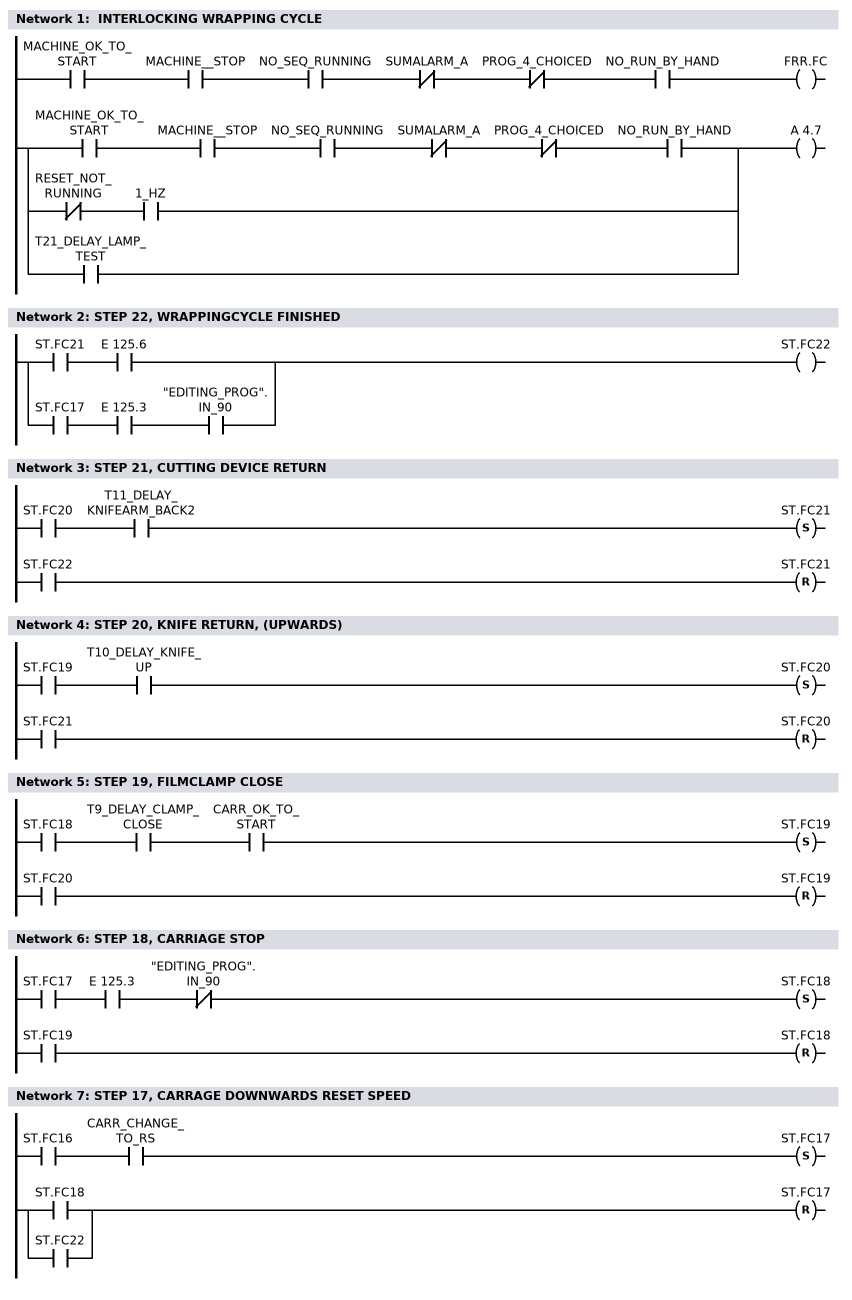
NETWORK
TITLE =  INTERLOCKING WRAPPING CYCLE
      A     "MACHINE_OK_TO_START";
      A     "MACHINE__STOP";
      A     "NO_SEQ_RUNNING";
      AN    "SUMALARM_A";
      AN    "PROG_4_CHOICED";
      A     "NO_RUN_BY_HAND";
      =     L 0.0;
      A     L 0.0;
      BLD   102;
      =     "FRR.FC";
      O     L 0.0;
      O;
      AN    "RESET_NOT_RUNNING";
      A     "1_HZ";
      O     "T21_DELAY_LAMP_TEST";
      =     "A 4.7";
NETWORK
TITLE = STEP 22, WRAPPINGCYCLE FINISHED
      A     "ST.FC21";
      A     "E 125.6";
      O;
      A     "ST.FC17";
      A     "E 125.3";
      A     "EDITING_PROG".IN_90;
      =     "ST.FC22";
NETWORK
TITLE = STEP 21, CUTTING DEVICE RETURN
      A     "ST.FC20";
      A     "T11_DELAY_KNIFEARM_BACK2";
      S     "ST.FC21";
      A     "ST.FC22";
      R     "ST.FC21";
      NOP   0;
NETWORK
TITLE = STEP 20, KNIFE RETURN, (UPWARDS)
      A     "ST.FC19";
      A     "T10_DELAY_KNIFE_UP";
      S     "ST.FC20";
      A     "ST.FC21";
      R     "ST.FC20";
      NOP   0;
NETWORK
TITLE = STEP 19, FILMCLAMP CLOSE
      A     "ST.FC18";
      A     "T9_DELAY_CLAMP_CLOSE";
      A     "CARR_OK_TO_START";
      S     "ST.FC19";
      A     "ST.FC20";
      R     "ST.FC19";
      NOP   0;
NETWORK
TITLE = STEP 18, CARRIAGE STOP
      A     "ST.FC17";
      A     "E 125.3";
      AN    "EDITING_PROG".IN_90;
      S     "ST.FC18";
      A     "ST.FC19";
      R     "ST.FC18";
      NOP   0;
NETWORK
TITLE = STEP 17, CARRAGE DOWNWARDS RESET SPEED
//STEG BEHÖVS EVENTUELT EJ????!!!!!!!!???????
      A     "ST.FC16";
      A     "CARR_CHANGE_TO_RS";
      S     "ST.FC17";
      A(;
      O     "ST.FC18";
      O     "ST.FC22";
      );
      R     "ST.FC17";
      NOP   0;
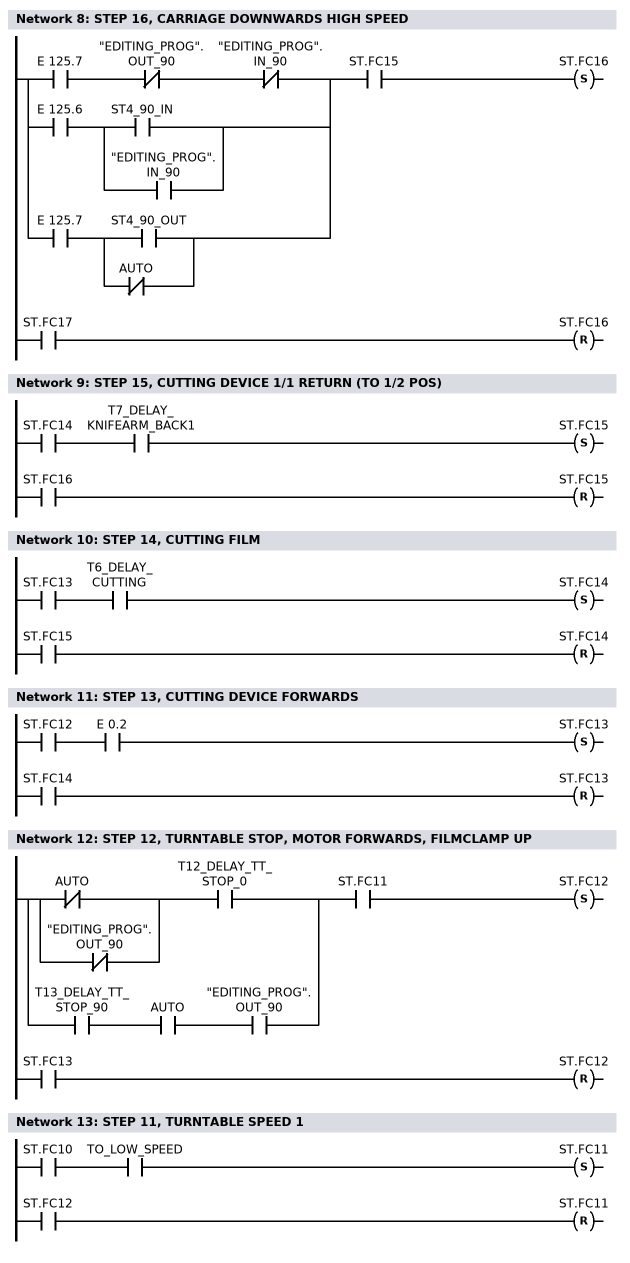
NETWORK
TITLE = STEP 16, CARRIAGE DOWNWARDS HIGH SPEED
      A(;
      A     "E 125.7";
      AN    "EDITING_PROG".OUT_90;
      AN    "EDITING_PROG".IN_90;
      O;
      A     "E 125.6";
      A(;
      O     "ST4_90_IN";
      O     "EDITING_PROG".IN_90;
      );
      O;
      A     "E 125.7";
      A(;
      O     "ST4_90_OUT";
      ON    "AUTO";
      );
      );
      A     "ST.FC15";
      S     "ST.FC16";
      A     "ST.FC17";
      R     "ST.FC16";
      NOP   0;
NETWORK
TITLE = STEP 15, CUTTING DEVICE 1/1 RETURN (TO 1/2 POS)
      A     "ST.FC14";
      A     "T7_DELAY_KNIFEARM_BACK1";
      S     "ST.FC15";
      A     "ST.FC16";
      R     "ST.FC15";
      NOP   0;
NETWORK
TITLE = STEP 14, CUTTING FILM
      A     "ST.FC13";
      A     "T6_DELAY_CUTTING";
      S     "ST.FC14";
      A     "ST.FC15";
      R     "ST.FC14";
      NOP   0;
NETWORK
TITLE = STEP 13, CUTTING DEVICE FORWARDS
      A     "ST.FC12";
      A     "E 0.2";
      S     "ST.FC13";
      A     "ST.FC14";
      R     "ST.FC13";
      NOP   0;
NETWORK
TITLE = STEP 12, TURNTABLE STOP, MOTOR FORWARDS, FILMCLAMP UP
      A(;
      A(;
      ON    "AUTO";
      ON    "EDITING_PROG".OUT_90;
      );
      A     "T12_DELAY_TT_STOP_0";
      O;
      A     "T13_DELAY_TT_STOP_90";
      A     "AUTO";
      A     "EDITING_PROG".OUT_90;
      );
      A     "ST.FC11";
      S     "ST.FC12";
      A     "ST.FC13";
      R     "ST.FC12";
      NOP   0;
NETWORK
TITLE = STEP 11, TURNTABLE SPEED 1
//STEG EV BORT ????????????
      A     "ST.FC10";
      A     "TO_LOW_SPEED";
      S     "ST.FC11";
      A     "ST.FC12";
      R     "ST.FC11";
      NOP   0;
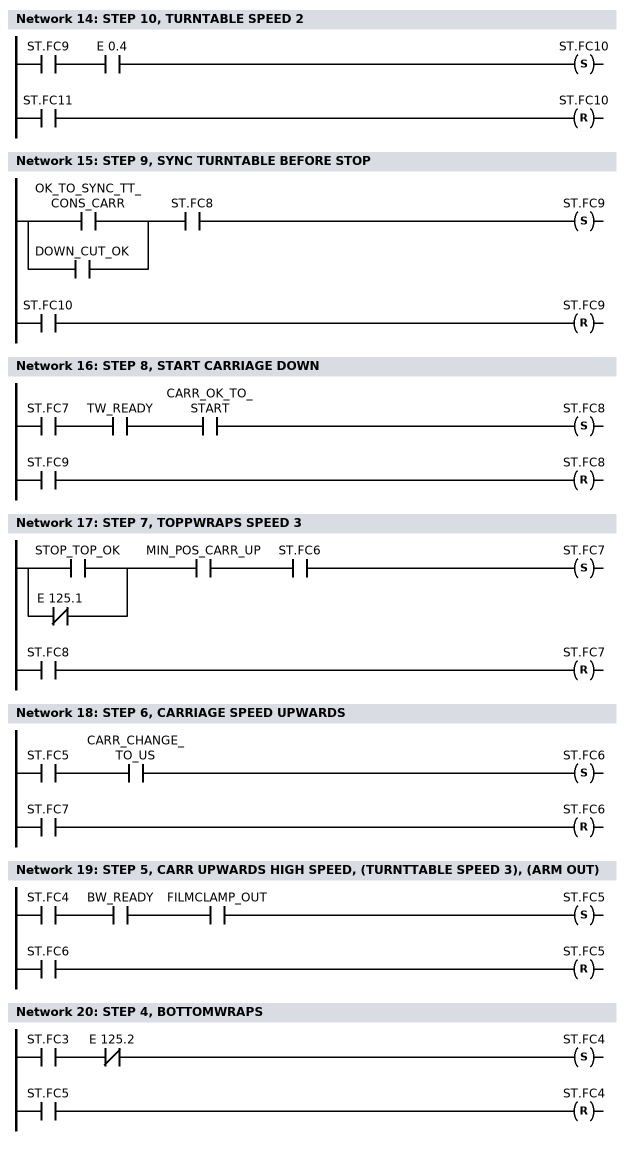
NETWORK
TITLE = STEP 10, TURNTABLE SPEED 2
      A     "ST.FC9";
      A     "E 0.4";
      S     "ST.FC10";
      A     "ST.FC11";
      R     "ST.FC10";
      NOP   0;
NETWORK
TITLE = STEP 9, SYNC TURNTABLE BEFORE STOP
//HISS STOPP, INTE OMRIKTARE TILL, MEN MÅSTE GÖRA NÅGOT FÖR ATT FÖRDRÖJA NGT 
//CYKEL VARV
//M 165.4 ej klart!!!!!!! skall ses över!!!!!!
      A(;
      O     "OK_TO_SYNC_TT_CONS_CARR";
      O     "DOWN_CUT_OK";
      );
      A     "ST.FC8";
      S     "ST.FC9";
      A     "ST.FC10";
      R     "ST.FC9";
      NOP   0;
NETWORK
TITLE = STEP 8, START CARRIAGE DOWN
      A     "ST.FC7";
      A     "TW_READY";
      A     "CARR_OK_TO_START";
      S     "ST.FC8";
      A     "ST.FC9";
      R     "ST.FC8";
      NOP   0;
NETWORK
TITLE = STEP 7, TOPPWRAPS SPEED 3
      A(;
      O     "STOP_TOP_OK";
      ON    "E 125.1";
      );
      A     "MIN_POS_CARR_UP";
      A     "ST.FC6";
      S     "ST.FC7";
      A     "ST.FC8";
      R     "ST.FC7";
      NOP   0;
NETWORK
TITLE = STEP 6, CARRIAGE SPEED UPWARDS
      A     "ST.FC5";
      A     "CARR_CHANGE_TO_US";
      S     "ST.FC6";
      A     "ST.FC7";
      R     "ST.FC6";
      NOP   0;
NETWORK
TITLE = STEP 5, CARR UPWARDS HIGH SPEED, (TURNTTABLE SPEED 3), (ARM OUT)
      A     "ST.FC4";
      A     "BW_READY";
      A     "FILMCLAMP_OUT";
      S     "ST.FC5";
      A     "ST.FC6";
      R     "ST.FC5";
      NOP   0;
NETWORK
TITLE = STEP 4, BOTTOMWRAPS
      A     "ST.FC3";
      AN    "E 125.2";
      S     "ST.FC4";
      A     "ST.FC5";
      R     "ST.FC4";
      NOP   0;
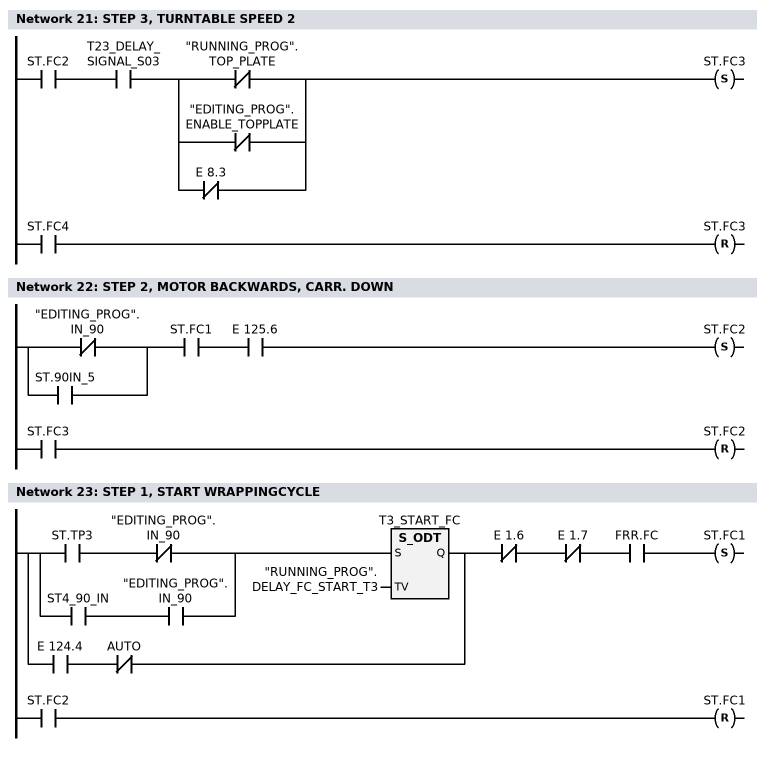
NETWORK
TITLE = STEP 3, TURNTABLE SPEED 2
      A     "ST.FC2";
      A     "T23_DELAY_SIGNAL_S03";
      A(;
      ON    "RUNNING_PROG".TOP_PLATE;
      ON    "EDITING_PROG".ENABLE_TOPPLATE;
      ON    "E 8.3";
      );
      S     "ST.FC3";
      A     "ST.FC4";
      R     "ST.FC3";
      NOP   0;
NETWORK
TITLE = STEP 2, MOTOR BACKWARDS, CARR. DOWN
      A(;
      ON    "EDITING_PROG".IN_90;
      O     "ST.90IN_5";
      );
      A     "ST.FC1";
      A     "E 125.6";
      S     "ST.FC2";
      A     "ST.FC3";
      R     "ST.FC2";
      NOP   0;
NETWORK
TITLE = STEP 1, START WRAPPINGCYCLE
      A(;
      O(;
      A(;
      A     "ST.TP3";
      AN    "EDITING_PROG".IN_90;
      O;
      A     "ST4_90_IN";
      A     "EDITING_PROG".IN_90;
      );
      L     "RUNNING_PROG".DELAY_FC_START_T3;
      SD    "T3_START_FC";
      NOP   0;
      NOP   0;
      NOP   0;
      A     "T3_START_FC";
      );
      O;
      A     "E 124.4";
      AN    "AUTO";
      );
      AN    "E 1.6";
      AN    "E 1.7";
      A     "FRR.FC";
      S     "ST.FC1";
      A     "ST.FC2";
      R     "ST.FC1";
      NOP   0;
END_FUNCTION

FUNCTION "START_AFTER_90_INFEED" : VOID	// FC 16
TITLE = HELP TO WRAPPING SEQ, START AFTER 90 DEGREE INFEEDING, OPTION
AUTHOR : LKA
NAME : START90I
VERSION : 0.0
BEGIN
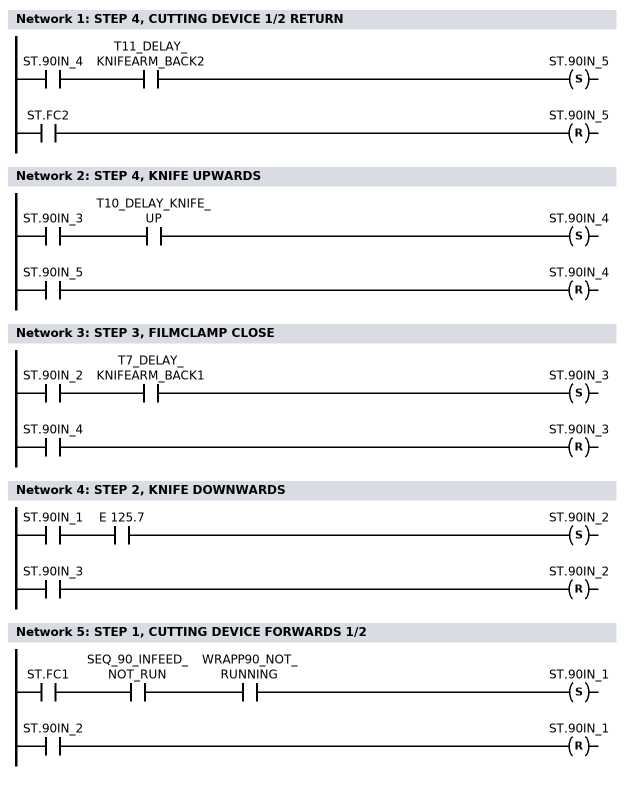
NETWORK
TITLE = STEP 4, CUTTING DEVICE 1/2 RETURN
//TID
      A     "ST.90IN_4";
      A     "T11_DELAY_KNIFEARM_BACK2";
      S     "ST.90IN_5";
      A     "ST.FC2";
      R     "ST.90IN_5";
      NOP   0;
NETWORK
TITLE = STEP 4, KNIFE UPWARDS
//TID
      A     "ST.90IN_3";
      A     "T10_DELAY_KNIFE_UP";
      S     "ST.90IN_4";
      A     "ST.90IN_5";
      R     "ST.90IN_4";
      NOP   0;
NETWORK
TITLE = STEP 3, FILMCLAMP CLOSE
//TID
      A     "ST.90IN_2";
      A     "T7_DELAY_KNIFEARM_BACK1";
      S     "ST.90IN_3";
      A     "ST.90IN_4";
      R     "ST.90IN_3";
      NOP   0;
NETWORK
TITLE = STEP 2, KNIFE DOWNWARDS
      A     "ST.90IN_1";
      A     "E 125.7";
      S     "ST.90IN_2";
      A     "ST.90IN_3";
      R     "ST.90IN_2";
      NOP   0;
NETWORK
TITLE = STEP 1, CUTTING DEVICE FORWARDS 1/2
      A     "ST.FC1";
      A     "SEQ_90_INFEED_NOT_RUN";
      A     "WRAPP90_NOT_RUNNING";
      S     "ST.90IN_1";
      A     "ST.90IN_2";
      R     "ST.90IN_1";
      NOP   0;
END_FUNCTION

FUNCTION "90_DEGREE_INFEED" : VOID	// FC 17
TITLE = 90 DEGREE INFEED, OPTION
AUTHOR : LKA
NAME : INF_90_D
VERSION : 0.1
BEGIN
